IF			BMP_Err.top AND
			Level_masla_Norm.top AND
			T_masla_Norm.top AND
			Krans_ready_to_move.top AND
			Krans_Poloj.top AND
			Net_AO_KC_SHKS04M.top AND
			Avt_SHU_vkl.top AND
			Nalichie220_SHU_Ai.top AND
			BP_Norm.top AND
			Naprajenie_U_IM.top AND
			//NOTAnalogNS.top AND 
			Not_AS.top AND
			dP_kr1.top AND
			Auto_Rej.top AND
			Impuls_Gaz.top AND ((algmanager.mode=modegpa.MODE_PUSKAP_R) OR (algmanager.mode=modegpa.MODE_PUSKPP_R) OR 
								(algmanager.mode=modegpa.MODE_PUSKAP_Ch) OR (algmanager.mode=modegpa.MODE_PUSKPP_Ch) OR
								(algmanager.mode=modegpa.MODE_I) OR (algmanager.mode=modegpa.MODE_PUSKK)) THEN
								ppuThird:=TRUE; ELSE ppuThird:=FALSE;	END_IF//ППУ для третьего этапа пуска
			

	IF		(NOT (im.kran6.so OR im.kran6.sz OR
			im.kran4.so OR im.kran4.sz)) AND
			(Im.kran6.onStatus=statusDualInput.STATUS_ON) AND 
			(Im.kran4.onStatus=statusDualInput.STATUS_ON) AND 
			Net_AO_KC_SHKS04M.top AND (NOT remont ()) AND
			(Im.kran1.onStatus=statusDualInput.STATUS_On) AND
			(Im.kran2.onStatus=statusDualInput.STATUS_On) AND
			Impuls_Gaz.top AND ((algmanager.mode=modegpa.MODE_PUSKAP_R) OR (algmanager.mode=modegpa.MODE_PUSKPP_R) OR 
								(algmanager.mode=modegpa.MODE_PUSKAP_Ch) OR (algmanager.mode=modegpa.MODE_PUSKPP_Ch) OR
								(algmanager.mode=modegpa.MODE_I) OR (algmanager.mode=modegpa.MODE_PUSKK)) THEN
								ppuForth:=TRUE; ELSE ppuForth:=FALSE; END_IF	//ППУ для четвертого этапа пуска

METHOD PUBLIC Neisp_DI : BOOL
VAR_INPUT
END_VAR
Neisp_DI:= 
		((ystavki.dPmg_Rassogl.status = 1) OR
		im.NalichieBP1_NS.Q OR
		im.NalichieBP2_NS.Q OR
		im.NalichieBP3_NS.Q OR
		im.NalichieBP4_NS.Q OR
		im.NalichieBP5_NS.Q OR
		im.NalichieBP6_NS.Q OR
		im.NalichieBP7_BP8_NS.Q OR
		im.NalichieBP9_BP10_NS.Q OR
		im.Nalichie_CU_MV_NS.Q OR
		im.Nalichie220BEAO_NS.Q OR
		im.NalichiePer220naVhode_NS.Q OR
		im.NalichiePost220naVhode_NS.Q OR
		im.NalichieBP11_NS.Q OR
		im.NalichieBP12_NS.Q OR
		im.NET_U_PNS.Q OR
		im.NET_U_CMN.Q OR
		im.NET_U_NU1.Q OR
		im.NET_U_NU2.Q OR
 		im.kran1.sdvig OR
		im.kran2.sdvig OR
		im.kran3.sdvig OR
		im.kran3b.sdvig OR
		im.kran4.sdvig OR
		im.kran5.sdvig OR
		im.kran6.sdvig OR
		(im.LevelMaslaAkkum.status = 1) OR
		im.MainRegOff.Q OR
		im.AVR_Vozb_Malfanctional.Q OR
		im.AsynchronnyHod.Q);
END_METHOD

METHOD PUBLIC analogsNs : BOOL
VAR_INPUT
END_VAR
VAR
		
END_VAR
SUPER^();
analogsNs:=
	
		(ai.TStalisStatoraKanall.interval 											< statusAi.NORMAL) 	OR
		(ai.TStalisStatoraKanal2.interval 											< statusAi.NORMAL) 	OR
		(ai.TStalisStatoraKanal3.interval 											< statusAi.NORMAL) 	OR
		(ai.TMediStatoraKanall.interval 											< statusAi.NORMAL) 	OR
		(ai.TMediStatoraKanal2.interval 											< statusAi.NORMAL) 	OR
		(ai.TMediStatoraKanal3.interval 											< statusAi.NORMAL) 	OR
		(ai.TOpornogoPodshipnikaEDT_1.interval 										< statusAi.NORMAL) 	OR
		(ai.TOpornoYpornogoPodshipnikaEDT_2.interval 								< statusAi.NORMAL) 	OR
		(ai.TOpornoYpornogoPodshipnikaKolesaRedEDT_3.interval 						< statusAi.NORMAL) 	OR
		(ai.TOpornoYpornogoPodshipnikaKolesaRedHT_4.interval 						< statusAi.NORMAL) 	OR
		(ai.TOpornogoPodshipnikaShesterniReduktoraT_5.interval 						< statusAi.NORMAL) 	OR
		(ai.TOpornogoPodshipnikaReduktoraHT_6.interval 								< statusAi.NORMAL) 	OR
		(ai.TOpornoYpornogoPodshipnikaNagnetateljaT_7_1.interval 					< statusAi.NORMAL) 	OR
		(ai.TOpornoYpornogoPodshipnikaNagnetateljaT_7_2.interval 					< statusAi.NORMAL) 	OR
		(ai.TOpornoYpornogoPodshipnikaSvobodnogoKoncaNT_8_1.interval 				< statusAi.NORMAL) 	OR
		(ai.TOpornoYpornogoPodshipnikaSvobodnogoKoncaNT_8_2.interval 				< statusAi.NORMAL) 	OR
		(ai.TYpornogoPodshipnikaRavKolodokHT_9_1.interval 							< statusAi.NORMAL) 	OR
		(ai.TYpornogoPodshipnikaRavKolodokHT_9_2.interval 							< statusAi.NORMAL) 	OR
		(ai.TYpornogoPodshipnikaNerabKolodokHT_10_1.interval 						< statusAi.NORMAL) 	OR
		(ai.TYpornogoPodshipnikaNerabKolodokHT_10_2.interval 						< statusAi.NORMAL) 	OR
		(ai.THolodnogoVozduhaEDKanall.interval 										< statusAi.NORMAL) 	OR
		(ai.THolodnogoVozduhaEDKanal2.interval 										< statusAi.NORMAL) 	OR
		(ai.TGorjachegoVozduhaEDKanall.interval 									< statusAi.NORMAL) 	OR
		(ai.TGorjachegoVozduhaEDKanal2.interval 									< statusAi.NORMAL) 	OR
		(ai.TgazaNaVhodeH.interval 													< statusAi.NORMAL) 	OR
		(ai.TgazaNaVyhodeH.interval 												< statusAi.NORMAL) 	OR
		(ai.TMasladoAVOM.interval 													< statusAi.NORMAL) 	OR
		(ai.TMaslaPosleAVOM.interval 												< statusAi.NORMAL) 	OR
		(ai.TMaslaMB.interval 														< statusAi.NORMAL) 	OR
		(ai.TMaslaMB_TEN.interval 													< statusAi.NORMAL) 	OR
		(ai.DavlenijaMasloSmNizkoe.interval 										< statusAi.NORMAL) 	OR
		(ai.PerepadDavlenieNaMasloFiltre.interval 									< statusAi.NORMAL) 	OR
		(ai.DavlenijaMasloSmVysokoe.interval 										< statusAi.NORMAL) 	OR
		(ai.DavlenijaMaslaPosleGNS.interval 										< statusAi.NORMAL) 	OR
		(ai.DavlenijaMaslaPosleNU.interval 											< statusAi.NORMAL) 	OR
		(ai.PerepadDavlenieNaKonfuzore.interval 									< statusAi.NORMAL) 	OR
		(ai.OsSdvigNagnetatelja_Plus.interval 										< statusAi.NORMAL) 	OR
		(ai.OsSdvigNagnetatelja_Minus.interval 										< statusAi.NORMAL) 	OR
		(ai.PerepadDavlenieMasloGaz.interval 										< statusAi.NORMAL) 	OR
		(ai.DGazaNaVhodeNagnetatelja.interval 										< statusAi.NORMAL) 	OR
		(ai.DGazaNaVyhodeNagnetatelja.interval 										< statusAi.NORMAL) 	OR
		(ai.DavlenieImpulsGaz.interval 												< statusAi.NORMAL) 	OR
		(ai.YrovenMaslaMB.interval 													< statusAi.NORMAL) 	OR
		(ai.Kontrol_per220V.interval 												< statusAi.NORMAL) 	OR
		(ai.Kontrol_post220V.interval 												< statusAi.NORMAL) 	OR
		(ai.VibroSkorostOPED_T1.interval 											< statusAi.NORMAL) 	OR
		(ai.VibroSkorostOYPED_T2.interval 											< statusAi.NORMAL) 	OR
		(ai.VibroSkorostOYPKolesaED_T3.interval 									< statusAi.NORMAL) 	OR
		(ai.VibroSkorostOPKolesaRH_T4.interval 										< statusAi.NORMAL) 	OR
		(ai.VibroSkorostOPShesterniRED_T5.interval 									< statusAi.NORMAL) 	OR
		(ai.VibroSkorostOPShesterniReduktoraH_T6.interval 							< statusAi.NORMAL) 	OR
		(ai.TokStatora.interval 													< statusAi.NORMAL) ;
END_METHOD

METHOD PRIVATE AS_PS_Anologs : BOOL
VAR_INPUT
END_VAR

 AS_PS_Anologs:= 	(ai.TMediStatoraKanall.interval 								= statusAi.NORMAL) 	AND 
 				 	(ai.TMediStatoraKanal2.interval 								= statusAi.NORMAL) 	AND
				 	(ai.TMediStatoraKanal3.interval 								= statusAi.NORMAL) 	AND
				 	(ai.TStalisStatoraKanall.interval 								= statusAi.NORMAL) 	AND
				 	(ai.TStalisStatoraKanal2.interval 								= statusAi.NORMAL) 	AND
				 	(ai.TStalisStatoraKanal3.interval 								= statusAi.NORMAL) 	AND
				 	(ai.TGorjachegoVozduhaEDKanall.interval 						= statusAi.NORMAL) 	AND
				 	(ai.TGorjachegoVozduhaEDKanal2.interval 						= statusAi.NORMAL) 	AND
				 	(ai.THolodnogoVozduhaEDKanall.interval 							= statusAi.NORMAL) 	AND
				 	(ai.THolodnogoVozduhaEDKanal2.interval 							= statusAi.NORMAL) 	AND
				 	(ai.TOpornogoPodshipnikaEDT_1.interval 							= statusAi.NORMAL) 	AND
					(ai.TOpornoYpornogoPodshipnikaEDT_2.interval 					= statusAi.NORMAL) 	AND
					(ai.TOpornoYpornogoPodshipnikaKolesaRedEDT_3.interval 			= statusAi.NORMAL) 	AND
					(ai.TOpornoYpornogoPodshipnikaKolesaRedHT_4.interval 			= statusAi.NORMAL) 	AND
					(ai.TOpornogoPodshipnikaShesterniReduktoraT_5.interval 			= statusAi.NORMAL) 	AND
					(ai.TOpornogoPodshipnikaReduktoraHT_6.interval 					= statusAi.NORMAL) 	AND
					(ai.TOpornoYpornogoPodshipnikaNagnetateljaT_7_1.interval 		= statusAi.NORMAL) 	AND
					(ai.TOpornoYpornogoPodshipnikaNagnetateljaT_7_2.interval 		= statusAi.NORMAL) 	AND
					(ai.TOpornoYpornogoPodshipnikaSvobodnogoKoncaNT_8_1.interval 	= statusAi.NORMAL) 	AND
					(ai.TOpornoYpornogoPodshipnikaSvobodnogoKoncaNT_8_2.interval 	= statusAi.NORMAL) 	AND
					(ai.TYpornogoPodshipnikaRavKolodokHT_9_1.interval 				= statusAi.NORMAL) 	AND
					(ai.TYpornogoPodshipnikaRavKolodokHT_9_2.interval 				= statusAi.NORMAL) 	AND
					(ai.TYpornogoPodshipnikaNerabKolodokHT_10_1.interval 			= statusAi.NORMAL) 	AND
					(ai.TYpornogoPodshipnikaNerabKolodokHT_10_2.interval 			= statusAi.NORMAL) 	AND
					(ai.TgazaNaVhodeH.interval 										= statusAi.NORMAL) 	AND
					(ai.TgazaNaVyhodeH.interval 									= statusAi.NORMAL) 	AND
					(ai.TMasladoAVOM.interval 										= statusAi.NORMAL) 	AND
					(ai.TMaslaPosleAVOM.interval 									= statusAi.NORMAL) 	AND
					(ai.TMaslaMB.interval 											= statusAi.NORMAL) 	AND
					(ai.TMaslaMB_TEN.interval 										= statusAi.NORMAL) 	AND			
					(ai.VibroSkorostOPED_T1.interval 								= statusAi.NORMAL) 	AND
					(ai.VibroSkorostOYPED_T2.interval 								= statusAi.NORMAL) 	AND
					(ai.VibroSkorostOYPKolesaED_T3.interval 						= statusAi.NORMAL) 	AND
					(ai.VibroSkorostOPKolesaRH_T4.interval 							= statusAi.NORMAL) 	AND
					(ai.VibroSkorostOPShesterniRED_T5.interval 						= statusAi.NORMAL) 	AND
					(ai.VibroSkorostOPShesterniReduktoraH_T6.interval 				= statusAi.NORMAL) 	AND
					(ai.OsSdvigNagnetatelja_Plus.interval 							= statusAi.NORMAL) 	AND
					(ai.OsSdvigNagnetatelja_Minus.interval 							= statusAi.NORMAL);
END_METHOD

METHOD PRIVATE haveAlarms : BOOL
VAR_INPUT
	
END_VAR

haveAlarms:= (NOT (Im.AOKC_SHKC.Q)) AND (im.AOKC_SHKC_CK.status = 1);
END_METHOD

METHOD PUBLIC reset
VAR_INPUT
END_VAR
SUPER^.reset();
ppuFirst_for_Pusk_Ch:=FALSE;
ppuFirst_for_Pusk_R:=FALSE;
ppuFirst_for_V_Ch:=FALSE;
ppuFirst_for_V_R:=FALSE;
ppuFirst_for_Pms_dPmg:=FALSE;
ppuFirst_for_K:=FALSE;
ppuFirst_for_I:=FALSE;
ppuSecond_V_Pusk_Ch:=FALSE;
ppuSecond_V_Pusk_R:=FALSE;
ppuSecond_I:=FALSE;
ppuThird:=FALSE;
ppuForth:=FALSE;
statusSet.setBit(15,FALSE); //к пуску готов
statusSet.setBit(16, FALSE); //к проверкам готов
statusSet.setBit(17,FALSE); //ко 2-му этапу пуска готов
statusSet.setBit(18,FALSE); //ко 3-му этапу пуска готов
statusSet.setBit(19,FALSE); //к 4-му этапу пуска готов
statusSet.setBit(20,FALSE); //к 4-му этапу пуска готов
END_METHOD

METHOD PUBLIC writeImStatus
VAR_INPUT
END_VAR
SUPER^.writeImStatus();

statusSet.setBit(15,ppuFirst_for_Pusk_Ch); //к пуску частотному
statusSet.setBit(16,ppuFirst_for_Pusk_r); //к пуску реакторному
statusSet.setBit(17,(ppuFirst_for_V_Ch OR ppuFirst_for_V_r OR ppuFirst_for_Pms_dPmg OR ppuFirst_for_K OR ppuFirst_for_I)); //к проверкам готов
statusSet.setBit(18,(ppuSecond_V_Pusk_ch OR ppuSecond_V_Pusk_r OR ppuSecond_I)); //ко 2-му этапу пуска готов
statusSet.setBit(19,(ppuThird)); //к 3-му этапу пуска готов
statusSet.setBit(20,(ppuForth)); //к 4-му этапу пуска готов
END_METHOD

METHOD public CK_Di : BOOL
VAR_INPUT
END_VAR

 CK_Di:=	(im.PerepadDavlenieMasloGaz_CK.status = 1)	AND
 			(im.PerepadDavlenieKran1_CK.status = 1)		AND
			(im.LevelMaslaAkkum_CK.status = 1)			AND
			(im.LoadDriveisGranted_CK.status = 1)		AND
			(im.VozbutetelisReady_CK.status = 1)			AND
			(im.RegVozbOff_CK.status = 1)				AND
			(im.MainRegOff_CK.status = 1)				AND
			(im.AVR_Vozb_Malfanctional_CK.status = 1)		AND
			(im.OFFAvarSwitch_CK.status = 1)				AND
			(im.AsynchronnyHod_CK.status = 1)		AND
			(im.Avtomat_SHU_on_CK.status = 1)		AND
			(im.Avtomat_SHP_on_CK.status = 1)			AND
			(im.U_Sekcii_CK.status = 1)					AND
			(im.Reactorni_Pusk_CK.status = 1)				AND
			(im.Chastotniy_Pusk_CK.status = 1)			AND
			(im.Fail_Chastotniy_Pusk_CK.status = 1)		AND
			(im.Hand_Reg_rej_CK.status = 1)				AND
			(im.AOKC_SHKC_CK.status = 1)					AND
			(im.NO_fromSHU_CK.status = 1)					AND
			(im.AO_fromSHU_CK.status = 1)					AND
			(im.AO_PRU_CK.status = 1)						AND
			(im.NKU_1_On_CK.status = 1)					AND
			(im.NKU_2_On_CK.status = 1)					AND
			(im.MVvkl_NAlichie_CK.status = 1)				AND
			(im.MVvykl_NAlichie_CK.status = 1)			AND
			(im.MVControl_Work_NAlichie_CK.status = 1)		AND
			(im.PNS_vkl_NAlichie_CK.status = 1)			AND
			(im.NU1_vkl_NAlichie_CK.status = 1)			AND
			(im.NU2_vkl_NAlichie_CK.status = 1)			AND
			(im.AVOM1_vkl_NAlichie_CK.status = 1)			AND
			(im.AVOM2_vkl_NAlichie_CK.status = 1)			AND
			(im.AVOM3_vkl_NAlichie_CK.status = 1)			AND
			(im.AVOM4_vkl_NAlichie_CK.status = 1)			AND
			(im.TEN_MB_vkl_NAlichie_CK.status = 1)			AND
			(im.TEN_Kollectora_vkl_NAlichie_CK.status = 1)	AND
			(im.Kalorifer_AVOM_vkl_NAlichie_CK.status = 1)	AND
			(im.CMN_vkl_NAlichie_CK.status = 1) AND (im.kran1.onstatus<>statusDualInput.STATUS_ERROR)
			AND (im.kran2.onstatus<>statusDualInput.STATUS_ERROR) AND (im.kran3.onstatus<>statusDualInput.STATUS_ERROR)
			AND (im.kran3b.onstatus<>statusDualInput.STATUS_ERROR) AND (im.kran4.onstatus<>statusDualInput.STATUS_ERROR)
			AND (im.kran5.onstatus<>statusDualInput.STATUS_ERROR)	AND (im.kran6.onstatus<>statusDualInput.STATUS_ERROR);
END_METHOD

METHOD PUBLIC Remont : BOOL
VAR_INPUT
END_VAR
Remont := protections.p_TOpornogoPodshipnikaEDT_1.remont OR

	
		
		protections.p_TOpornoYpornogoPodshipnikaEDT_2.remont OR
		protections.p_TOpornoYpornogoPodshipnikaKolesaRedEDT_3.remont OR
		protections.p_TOpornoYpornogoPodshipnikaKolesaRedHT_4.remont OR
		protections.p_TOpornogoPodshipnikaShesterniReduktoraT_5.remont OR
		protections.p_TOpornogoPodshipnikaReduktoraHT_6.remont OR
		protections.p_TOpornoYpornogoPodshipnikaNagnetateljaT_7.remont OR
		protections.p_TOpornoYpornogoPodshipnikaSvobodnogoKoncaNT_8.remont OR
		protections.p_TYpornogoPodshipnikaRavKolodokHT_9.remont OR
		protections.p_TYpornogoPodshipnikaNerabKolodokHT_10.remont OR
		protections.p_TgazaNaVyhodeH.remont OR
		
	(*Давления*)
		
		protections.p_OsSdvigNagnetatelja_Plus.remont OR
		protections.p_OsSdvigNagnetatelja_Minus.remont OR
		protections.p_DGazaNaVhodeNagnetatelja_GPA_STOP.remont OR
		protections.p_DGazaNaVyhodeNagnetatelja_GPA_STOP.remont OR
		//protections.p_DGazaNaVhodeNagnetatelja.remont OR
		protections.p_DGazaNaVyhodeNagnetatelja.remont OR
		protections.p_PerepadDavlenieMasloGaz.remont OR
		protections.p_DavlenijaMasloSmNizkoe.remont OR
		protections.p_DavlenijaMasloSmVysokoe.remont OR
	
	(*Вибрация*)
		
		protections.p_VibroSkorostOPED_T1.remont OR
		protections.p_VibroSkorostOYPED_T2.remont OR
		protections.p_VibroSkorostOYPKolesaED_T3.remont OR
		protections.p_VibroSkorostOPKolesaRH_T4.remont OR
		protections.p_VibroSkorostOPShesterniRED_T5.remont OR
		protections.p_VibroSkorostOPShesterniReduktoraH_T6.remont OR
	(*Дискретные сигналы *)
		
		protections.p_PerepadDavlenieMasloGaz_Less100.remont OR
		protections.p_RegVozbOff.remont OR
		protections.p_Fail_Chastotniy_Pusk.remont OR
		protections.p_OFFAvarSwitch.remont OR
		protections.p_AOKC_SHKC.remont OR
		protections.p_AO_PRU.remont OR
		protections.p_AO_fromSHU.remont OR	
					
(*Защиты по ИМ *)																							
		protections.p_mvOff.remont OR
		protections.p_kran1.remont OR
		protections.p_kran2.remont;
END_METHOD

END_FUNCTION_BLOCK

// K1/std12k5/Pusk/puskFirst_faza1
	{attribute 'symbol' := 'none'}
FUNCTION_BLOCK puskFirst_faza1 EXTENDS StepBySteapAlgoritm
VAR_INPUT
	
END_VAR
VAR_OUTPUT
END_VAR
VAR
	{attribute 'symbol' := 'read'}
	timer240:		ph_Timer (table:=ADR(phasesTable)):=		(phaseNumber:=0, delay:=T#240S);
	pnsOn:			ph_Switch (table:=ADR(phasesTable)):=		(phaseNumber:=1, Im:=Im.pns, act:=DualStateImAction.on);
	psmMore50:		CustomPhase (table:=ADR(phasesTable)):=		(phaseNumber:=2);
	psmMore300:		CustomPhase (table:=ADR(phasesTable)):=		(phaseNumber:=3);
	Protection_Pms: CustomPhase (table:=ADR(phasesTable)):=		(phaseNumber:=4);
	Error_Alg:		CustomPhase (table:=ADR(phasesTable)):=		(phaseNumber:=5);
END_VAR

SUPER^();
IF 	NOT Protection_Pms.top THEN
	timer240.run (); //запускаем таймер включаем ПНС
END_IF;
IF NOT pnsON.start THEN
	pnsOn.run();
END_IF
///////////////////////////////////////////////////////
IF 	pnsOn.top THEN //ПНС включен и таймер не истек
	psmMore50.run(); //запускаем проверку условия Pмс >50 
	psmMore300.run(); //запускаем проверку условия Pмс >300 
END_IF
///////////////////////////////////////////////////////
IF	psmMore50.start AND (NOT psmMore50.top) THEN
	IF 	ai.DavlenijaMasloSmNizkoe.interval>=statusAi.NORMAL AND ai.DavlenijaMasloSmNizkoe.value > 50  THEN
	  	psmMore50.top:=TRUE;
	END_IF
END_IF
///////////////////////////////////////////////////////
IF  psmMore300.start AND (NOT psmMore300.top) THEN
	IF 	ai.DavlenijaMasloSmVysokoe.interval>=statusAi.NORMAL AND ai.DavlenijaMasloSmVysokoe.value > 300  THEN
	  	psmMore300.top:=TRUE;
	END_IF	
END_IF
///////////////////////////////////////////////////////
IF	psmMore50.top AND psmMore300.top THEN
	Protection_Pms.run ();
END_IF
///////////////////////////////////////////////////////
IF	Protection_Pms.start AND (NOT Protection_Pms.top) THEN //защита по давлению масла смазки включить
	protections.p_DavlenijaMasloSmNizkoe.run();
	protections.p_DavlenijaMasloSmVysokoe.run ();
	Protection_Pms.top := TRUE;
END_IF
///////////////////////////////////////////////////////
IF	timer240.top THEN //Ошибка завершения алгоритма по таймеру
	Error_Alg.ERROR := TRUE;
ELSE
	Error_Alg.ERROR := FALSE;	
END_IF
///////////////////////////////////////////////////////
IF	Protection_Pms.top THEN
	timer240.reset();
	end ();
END_IF
///////////////////////////////////////////////////////

METHOD PUBLIC reset
VAR_INPUT
END_VAR
SUPER^.reset();
statusSet.setBit(15,0);
END_METHOD

METHOD PUBLIC run
VAR_INPUT
END_VAR
SUPER^.run();
statusSet.setBit(15,1);
END_METHOD

END_FUNCTION_BLOCK

// K2/std12k5/Pusk/puskFirst_faza1
	{attribute 'symbol' := 'none'}
FUNCTION_BLOCK puskFirst_faza1 EXTENDS StepBySteapAlgoritm
VAR_INPUT
	
END_VAR
VAR_OUTPUT
END_VAR
VAR
	{attribute 'symbol' := 'read'}
	timer240:		ph_Timer (table:=ADR(phasesTable)):=		(phaseNumber:=0, delay:=T#240S);
	pnsOn:			ph_Switch (table:=ADR(phasesTable)):=		(phaseNumber:=1, Im:=Im.pns, act:=DualStateImAction.on);
	psmMore50:		CustomPhase (table:=ADR(phasesTable)):=		(phaseNumber:=2);
	psmMore300:		CustomPhase (table:=ADR(phasesTable)):=		(phaseNumber:=3);
	Protection_Pms: CustomPhase (table:=ADR(phasesTable)):=		(phaseNumber:=4);
	Error_Alg:		CustomPhase (table:=ADR(phasesTable)):=		(phaseNumber:=5);
END_VAR

SUPER^();
IF 	NOT Protection_Pms.top THEN
	timer240.run (); //запускаем таймер включаем ПНС
END_IF;
IF NOT pnsON.start THEN
	pnsOn.run();
END_IF
///////////////////////////////////////////////////////
IF 	pnsOn.top THEN //ПНС включен и таймер не истек
	psmMore50.run(); //запускаем проверку условия Pмс >50 
	psmMore300.run(); //запускаем проверку условия Pмс >300 
END_IF
///////////////////////////////////////////////////////
IF	psmMore50.start AND (NOT psmMore50.top) THEN
	IF 	ai.DavlenijaMasloSmNizkoe.interval>=statusAi.NORMAL AND ai.DavlenijaMasloSmNizkoe.value > 50  THEN
	  	psmMore50.top:=TRUE;
	END_IF
END_IF
///////////////////////////////////////////////////////
IF  psmMore300.start AND (NOT psmMore300.top) THEN
	IF 	ai.DavlenijaMasloSmVysokoe.interval>=statusAi.NORMAL AND ai.DavlenijaMasloSmVysokoe.value > 300  THEN
	  	psmMore300.top:=TRUE;
	END_IF	
END_IF
///////////////////////////////////////////////////////
IF	psmMore50.top AND psmMore300.top THEN
	Protection_Pms.run ();
END_IF
///////////////////////////////////////////////////////
IF	Protection_Pms.start AND (NOT Protection_Pms.top) THEN //защита по давлению масла смазки включить
	protections.p_DavlenijaMasloSmNizkoe.run();
	protections.p_DavlenijaMasloSmVysokoe.run ();
	Protection_Pms.top := TRUE;
END_IF
///////////////////////////////////////////////////////
IF	timer240.top THEN //Ошибка завершения алгоритма по таймеру
	Error_Alg.ERROR := TRUE;
ELSE
	Error_Alg.ERROR := FALSE;	
END_IF
///////////////////////////////////////////////////////
IF	Protection_Pms.top THEN
	timer240.reset();
	end ();
END_IF
///////////////////////////////////////////////////////

METHOD PUBLIC reset
VAR_INPUT
END_VAR
SUPER^.reset();
statusSet.setBit(15,0);
END_METHOD

METHOD PUBLIC run
VAR_INPUT
END_VAR
SUPER^.run();
statusSet.setBit(15,1);
END_METHOD

END_FUNCTION_BLOCK

// K1/std12k5/Pusk/puskFirst_faza2
	{attribute 'symbol' := 'none'}
FUNCTION_BLOCK puskFirst_faza2 EXTENDS StepBySteapAlgoritm
VAR_INPUT
	
END_VAR
VAR_OUTPUT
END_VAR
VAR
	{attribute 'symbol' := 'read'}
	timer240:		ph_Timer 	(table:=ADR(phasesTable)):=		(phaseNumber:=0, delay:=T#240S);
	nuOn:			CustomPhase (table:=ADR(phasesTable)):=		(phaseNumber:=1);
	dPmg_more100:	CustomPhase (table:=ADR(phasesTable)):=		(phaseNumber:=2);
	Error_Alg:		CustomPhase (table:=ADR(phasesTable)):=		(phaseNumber:=3);
	Auto_NU1:		CustomPhase (table:=ADR(phasesTable)):=		(phaseNumber:=4);
END_VAR

SUPER^();
IF 	NOT dPmg_more100.top THEN
	timer240.run (); //запускаем таймер включаем ПНС
END_IF
IF	NOT nuon.start THEN
	nuOn.run();
END_IF
///////////////////////////////////////////////////////
IF 	nuOn.start AND NOT nuOn.top THEN //НУ включен
	CASE 	im.nu.mainNasos.Value OF
	0:		im.nu.nu1.on ();
	1:		im.nu.nu2.on ();
	END_CASE
END_IF
///////////////////////////////////////////////////////
IF	((im.nu.nu1.onStatus = statusDualInput.status_on) OR (im.nu.nu2.onStatus = statusDualInput.status_on)) AND  nuOn.start THEN
	dPmg_more100.run(); //запускаем проверку условия dPmg_more100
	nuOn.top:=TRUE;
END_IF
///////////////////////////////////////////////////////
IF	dPmg_more100.start AND (NOT dPmg_more100.top) THEN
	IF 	(NOT im.PerepadDavlenieMasloGaz_Less100.Q) AND (im.PerepadDavlenieMasloGaz_CK.status = 1) AND 
		(ai.PerepadDavlenieMasloGaz.interval	>=	statusAi.NORMAL) AND (ai.PerepadDavlenieMasloGaz.value > 150) THEN
	  	dPmg_more100.top:=TRUE;
	END_IF
END_IF
///////////////////////////////////////////////////////
IF	timer240.top THEN //Ошибка завершения алгоритма по таймеру
	Error_Alg.ERROR := TRUE;
ELSE
	Error_Alg.ERROR := FALSE;	
END_IF
///////////////////////////////////////////////////////
IF	dPmg_more100.top AND nuOn.top THEN
	Auto_NU1.top:=TRUE;
	protections.p_PerepadDavlenieMasloGaz.run();
	protections.p_PerepadDavlenieMasloGaz_Less100.run ();
	protections.p_DGazaNaVhodeNagnetatelja_GPA_STOP.reset ();
	protections.p_DGazaNaVyhodeNagnetatelja_GPA_STOP.reset ();
	algoritms.autoNu_1.CanRun:=TRUE;
	algoritms.autoNu_1.run ();
	timer240.reset();
	end();
END_IF

END_FUNCTION_BLOCK

// K2/std12k5/Pusk/puskFirst_faza2
	{attribute 'symbol' := 'none'}
FUNCTION_BLOCK puskFirst_faza2 EXTENDS StepBySteapAlgoritm
VAR_INPUT
	
END_VAR
VAR_OUTPUT
END_VAR
VAR
	{attribute 'symbol' := 'read'}
	timer240:		ph_Timer 	(table:=ADR(phasesTable)):=		(phaseNumber:=0, delay:=T#240S);
	nuOn:			CustomPhase (table:=ADR(phasesTable)):=		(phaseNumber:=1);
	dPmg_more100:	CustomPhase (table:=ADR(phasesTable)):=		(phaseNumber:=2);
	Error_Alg:		CustomPhase (table:=ADR(phasesTable)):=		(phaseNumber:=3);
	Auto_NU1:		CustomPhase (table:=ADR(phasesTable)):=		(phaseNumber:=4);
END_VAR

SUPER^();
IF 	NOT dPmg_more100.top THEN
	timer240.run (); //запускаем таймер включаем ПНС
END_IF;
IF	NOT nuon.start THEN
	nuOn.run();
END_IF
///////////////////////////////////////////////////////
IF 	nuOn.start AND NOT nuOn.top THEN //НУ включен
	CASE 	im.nu.mainNasos.Value OF
	0:		im.nu.nu1.on ();
	1:		im.nu.nu2.on ();
	END_CASE
END_IF
///////////////////////////////////////////////////////
IF	((im.nu.nu1.onStatus = statusDualInput.status_on) OR (im.nu.nu2.onStatus = statusDualInput.status_on)) AND  nuOn.start THEN
	dPmg_more100.run(); //запускаем проверку условия dPmg_more100
	nuOn.top:=TRUE;
END_IF
///////////////////////////////////////////////////////
IF	dPmg_more100.start AND (NOT dPmg_more100.top) THEN
	IF 	(NOT im.PerepadDavlenieMasloGaz_Less100.Q) AND (im.PerepadDavlenieMasloGaz_CK.status = 1) AND 
		(ai.PerepadDavlenieMasloGaz.interval	>=	statusAi.NORMAL) AND (ai.PerepadDavlenieMasloGaz.value > 150) THEN
	  	dPmg_more100.top:=TRUE;
	END_IF
END_IF
///////////////////////////////////////////////////////
IF	timer240.top THEN //Ошибка завершения алгоритма по таймеру
	Error_Alg.ERROR := TRUE;
ELSE
	Error_Alg.ERROR := FALSE;	
END_IF
///////////////////////////////////////////////////////
IF	dPmg_more100.top AND nuOn.top THEN
	Auto_NU1.top:=TRUE;
	protections.p_PerepadDavlenieMasloGaz.run();
	protections.p_PerepadDavlenieMasloGaz_Less100.run ();
	protections.p_DGazaNaVhodeNagnetatelja_GPA_STOP.reset ();
	protections.p_DGazaNaVyhodeNagnetatelja_GPA_STOP.reset ();
	algoritms.autoNu_1.CanRun:=TRUE;
	algoritms.autoNu_1.run ();
	timer240.reset();
	end();
END_IF

END_FUNCTION_BLOCK

// K1/std12k5/Pusk/puskSecond_faza_Reactor
{attribute 'symbol' := 'none'}
FUNCTION_BLOCK puskSecond_faza_Reactor EXTENDS StepBySteapAlgoritm
VAR_INPUT
	autoAVOM_canrun_flag:BOOL;
END_VAR
VAR_OUTPUT
	
END_VAR
VAR
	{attribute 'symbol' := 'read'}
	timer25:			ph_Timer (table:=ADR(phasesTable)):=		(phaseNumber:=0, delay:=T#25S);
	{attribute 'symbol' := 'read'}
	timer3:				ph_Timer (table:=ADR(phasesTable)):=		(phaseNumber:=1, delay:=T#3S);
	mvOn:				ph_Switch (table:=ADR(phasesTable)):=		(phaseNumber:=2, Im:=Im.mv, act:=DualStateImAction.on);
	pGNSmore04:			CustomPhase (table:=ADR(phasesTable)):=		(phaseNumber:=3);
	gotov_K_zagruzke: 	ph_SingleSignal (table:=ADR(phasesTable)):=	(phaseNumber:=4, im:=im.LoadDriveisGranted, expectedValue:=TRUE);
	
	dPmg_Top:			CustomPhase (table:=ADR(phasesTable)):=		(phaseNumber:=6);
	
	Mv_Error:			CustomPhase (table:=ADR(phasesTable)):=		(phaseNumber:=8);
	AutoPNS_start:		CustomPhase (table:=ADR(phasesTable)):=		(phaseNumber:=9);
END_VAR

SUPER^();
IF 	NOT mvOn.top THEN
	timer25.run (); //запускаем таймер 25 сек
END_IF
IF	NOT mvOn.top THEN
	timer3.run (); //запускаем таймер 3 сек
END_IF
IF	NOT mvOn.start THEN
	mvOn.run();
END_IF
///////////////////////////////////////////////////////
IF 	mvOn.top  THEN 
	IF	NOT pGNSmore04.start AND ((algManager.mode = modegpa.MODE_PUSKAP_R) OR (algManager.mode = modegpa.MODE_PUSKPP_R)) THEN //проверяем условие по давление за ГНС > 400 кПа
		pGNSmore04.run(); 
	END_IF
	IF	NOT autoAVOM_canrun_flag THEN
		algoritms.S_AutoAVOM.CanRun:=TRUE;
		autoAVOM_canrun_flag:=TRUE;
	END_IF
	timer3.reset ();
	timer25.reset ();
	Mv_Error.error := FALSE;
	gotov_K_zagruzke.run();
	IF	(NOT dPmg_Top.start) AND ((algManager.mode = modegpa.MODE_PUSKAP_R) OR (algManager.mode = modegpa.MODE_PUSKPP_R)) THEN
		dPmg_Top.run ();
	END_IF
	protections.p_mvOff.run (); //включаем защиты по МВ и возбудителю
	protections.p_OFFAvarSwitch.run();
	protections.p_RegVozbOff.run();
ELSIF	NOT mvOn.top AND timer3.top THEN
		Mv_Error.error := TRUE;
END_IF

///////////////////////////////////////////////////////
IF	dPmg_Top.start AND (NOT dPmg_Top.top) THEN
	IF	(NOT im.PerepadDavlenieMasloGaz_Less100.Q) AND (im.PerepadDavlenieMasloGaz_CK.status = 1) AND (ai.PerepadDavlenieMasloGaz.value > 150)	THEN //по аналогу проверяем только значение, т.к. при пуске может уйти в зашкал
		dPmg_Top.top:=TRUE;
		protections.p_PerepadDavlenieMasloGaz.run();
		protections.p_PerepadDavlenieMasloGaz_Less100.run ();
		protections.p_DGazaNaVhodeNagnetatelja_GPA_STOP.reset ();
		protections.p_DGazaNaVyhodeNagnetatelja_GPA_STOP.reset ();
		algoritms.autoNu_2.CanRun:=TRUE;
		algoritms.autoNu_2.run ();
	END_IF
END_IF
///////////////////////////////////////////////////////
IF	pGNSmore04.start AND (NOT pGNSmore04.top) THEN //Давление после ГНС больше 400 кПА
	IF 	(ai.DavlenijaMaslaPosleGNS.interval	>=statusAi.NORMAL) AND (ai.DavlenijaMaslaPosleGNS.value	 > 400) THEN
	  	pGNSmore04.top:=TRUE; 
	END_IF
END_IF
///////////////////////////////////////////////////////
IF	((pGNSmore04.top AND gotov_K_zagruzke.top AND dPmg_Top.top AND ((algManager.mode = modegpa.MODE_PUSKAP_R) OR (algManager.mode = modegpa.MODE_PUSKPP_R))) OR 
	(gotov_K_zagruzke.top AND ((algManager.mode = modegpa.MODE_PUSKV_R) OR (algManager.mode = modegpa.MODE_I)))) AND NOT AutoPNS_start.top  THEN 
	algoritms.AutoPNS_Start.CanRun :=TRUE;
	algoritms.AutoPNS_Start.run();
	AutoPNS_start.top:=TRUE;
	end();
END_IF
IF	timer25.top AND Mv_Error.error THEN
	algoritms.ao.CanRun:=TRUE;
	algoritms.ao.run ();
	
END_IF

METHOD PUBLIC reset
VAR_INPUT
END_VAR
SUPER^.reset();
statusSet.setBit(15,0);
END_METHOD

METHOD PUBLIC run
VAR_INPUT
END_VAR
SUPER^.run();
statusSet.setBit(15,1);
END_METHOD

END_FUNCTION_BLOCK

// K2/std12k5/Pusk/puskSecond_faza_Reactor
{attribute 'symbol' := 'none'}
FUNCTION_BLOCK puskSecond_faza_Reactor EXTENDS StepBySteapAlgoritm
VAR_INPUT
	autoAVOM_canrun_flag:BOOL;
END_VAR
VAR_OUTPUT
	
END_VAR
VAR
	{attribute 'symbol' := 'read'}
	timer25:			ph_Timer (table:=ADR(phasesTable)):=		(phaseNumber:=0, delay:=T#25S);
	{attribute 'symbol' := 'read'}
	timer3:				ph_Timer (table:=ADR(phasesTable)):=		(phaseNumber:=1, delay:=T#3S);
	mvOn:				ph_Switch (table:=ADR(phasesTable)):=		(phaseNumber:=2, Im:=Im.mv, act:=DualStateImAction.on);
	pGNSmore04:			CustomPhase (table:=ADR(phasesTable)):=		(phaseNumber:=3);
	gotov_K_zagruzke: 	ph_SingleSignal (table:=ADR(phasesTable)):=	(phaseNumber:=4, im:=im.LoadDriveisGranted, expectedValue:=TRUE);
	
	dPmg_Top:			CustomPhase (table:=ADR(phasesTable)):=		(phaseNumber:=6);
	
	Mv_Error:			CustomPhase (table:=ADR(phasesTable)):=		(phaseNumber:=8);
	AutoPNS_start:		CustomPhase (table:=ADR(phasesTable)):=		(phaseNumber:=9);
END_VAR

SUPER^();
IF 	NOT mvOn.top THEN
	timer25.run (); //запускаем таймер 25 сек
END_IF
IF	NOT mvOn.top THEN
	timer3.run (); //запускаем таймер 3 сек
END_IF
IF	NOT mvOn.start THEN
	mvOn.run();
END_IF
///////////////////////////////////////////////////////
IF 	mvOn.top  THEN 
	IF	NOT pGNSmore04.start AND ((algManager.mode = modegpa.MODE_PUSKAP_R) OR (algManager.mode = modegpa.MODE_PUSKPP_R)) THEN //проверяем условие по давление за ГНС > 400 кПа
		pGNSmore04.run(); 
	END_IF
	IF	NOT autoAVOM_canrun_flag THEN
		algoritms.S_AutoAVOM.CanRun:=TRUE;
		autoAVOM_canrun_flag:=TRUE;
	END_IF
	timer3.reset ();
	timer25.reset ();
	Mv_Error.error := FALSE;
	gotov_K_zagruzke.run();
	IF	(NOT dPmg_Top.start) AND ((algManager.mode = modegpa.MODE_PUSKAP_R) OR (algManager.mode = modegpa.MODE_PUSKPP_R)) THEN
		dPmg_Top.run ();
	END_IF
	protections.p_mvOff.run (); //включаем защиты по МВ и возбудителю
	protections.p_OFFAvarSwitch.run();
	protections.p_RegVozbOff.run();
ELSIF	NOT mvOn.top AND timer3.top THEN
		Mv_Error.error := TRUE;
END_IF

///////////////////////////////////////////////////////
IF	dPmg_Top.start AND (NOT dPmg_Top.top) THEN
	IF	(NOT im.PerepadDavlenieMasloGaz_Less100.Q) AND (im.PerepadDavlenieMasloGaz_CK.status = 1)AND (ai.PerepadDavlenieMasloGaz.value > 150)	THEN //по аналогу проверяем только значение, т.к. при пуске может уйти в зашкал
		dPmg_Top.top:=TRUE;
		protections.p_PerepadDavlenieMasloGaz.run();
		protections.p_PerepadDavlenieMasloGaz_Less100.run ();
		protections.p_DGazaNaVhodeNagnetatelja_GPA_STOP.reset ();
		protections.p_DGazaNaVyhodeNagnetatelja_GPA_STOP.reset ();
		algoritms.autoNu_2.CanRun:=TRUE;
		algoritms.autoNu_2.run ();
	END_IF
END_IF
///////////////////////////////////////////////////////
IF	pGNSmore04.start AND (NOT pGNSmore04.top) THEN //Давление после ГНС больше 400 кПА
	IF 	(ai.DavlenijaMaslaPosleGNS.interval	>=statusAi.NORMAL) AND (ai.DavlenijaMaslaPosleGNS.value	 > 400) THEN
	  	pGNSmore04.top:=TRUE; 
	END_IF
END_IF
///////////////////////////////////////////////////////
IF	((pGNSmore04.top AND gotov_K_zagruzke.top AND dPmg_Top.top AND ((algManager.mode = modegpa.MODE_PUSKAP_R) OR (algManager.mode = modegpa.MODE_PUSKPP_R))) OR 
	(gotov_K_zagruzke.top AND ((algManager.mode = modegpa.MODE_PUSKV_R) OR (algManager.mode = modegpa.MODE_I)))) AND NOT AutoPNS_start.top  THEN 
	algoritms.AutoPNS_Start.CanRun :=TRUE;
	algoritms.AutoPNS_Start.run();
	AutoPNS_start.top:=TRUE;
	end();
END_IF
IF	timer25.top AND Mv_Error.error THEN
	algoritms.ao.CanRun:=TRUE;
	algoritms.ao.run ();
	
END_IF

METHOD PUBLIC reset
VAR_INPUT
END_VAR
SUPER^.reset();
statusSet.setBit(15,0);
END_METHOD

METHOD PUBLIC run
VAR_INPUT
END_VAR
SUPER^.run();
statusSet.setBit(15,1);
END_METHOD

END_FUNCTION_BLOCK

// K1/std12k5/Pusk/puskThird_faza
	{attribute 'symbol' := 'none'}
FUNCTION_BLOCK puskThird_faza EXTENDS StepBySteapAlgoritm
VAR_INPUT
	Smazka_1_2:BOOL;
END_VAR
VAR_OUTPUT
	
END_VAR
VAR
	{attribute 'symbol' := 'read'}
	timer480:		ph_Timer (table:=ADR(phasesTable)):=		(phaseNumber:=0, delay:=T#480S);
	kran4Open:		CustomPhase (table:=ADR(phasesTable)):=		(phaseNumber:=1);
	{attribute 'symbol' := 'read'}
	waitAfterKran4:	ph_Timer (table:=ADR(phasesTable)):=		(phaseNumber:=2, delay:=T#10S);
	kran5Close:		ph_Kran (table:=ADR(phasesTable)):=			(phaseNumber:=3, Im:=Im.kran5, act:=DualStateImAction.off);	
	kran3bOpen:		CustomPhase (table:=ADR(phasesTable)):=		(phaseNumber:=4);
	dP_kr1less100: 	ph_SingleSignal (table:=ADR(phasesTable)):=	(phaseNumber:=5, im:=Im.PerepadDavlenieKran1_Less100, expectedValue:=TRUE);
	Pvh_vyhMore5:	CustomPhase (table:=ADR(phasesTable)):=		(phaseNumber:=6);
	kran1Open:		ph_Kran (table:=ADR(phasesTable)):=			(phaseNumber:=7, Im:=Im.kran1, act:=DualStateImAction.on);	
	kran2Open:		ph_Kran (table:=ADR(phasesTable)):=			(phaseNumber:=8, Im:=Im.kran2, act:=DualStateImAction.on);
	kran3Open:		ph_Kran (table:=ADR(phasesTable)):=			(phaseNumber:=9, Im:=Im.kran3, act:=DualStateImAction.on);
	kran3bClose:	ph_Kran (table:=ADR(phasesTable)):=			(phaseNumber:=10, Im:=Im.kran3b, act:=DualStateImAction.off);
	Err_ALG:		CustomPhase (table:=ADR(phasesTable)):=		(phaseNumber:=11);
END_VAR

SUPER^();
IF	NOT (kran3bClose.top) THEN
	timer480.run (); //запускаем таймер 480 секунд
END_IF;
////////////////////***Открываем кран 4****//////////////////////////
IF	NOT kran1Open.top AND im.kran4._cmdreset.IN = FALSE  THEN
	
	im.Kr_4_Open_From_Alg.on();
	kran4Open.run();
END_IF;
IF	kran4Open.start AND NOT kran4Open.top THEN
	IF	im.kran4.onStatus = statusDualInput.STATUS_ON THEN
		kran4Open.top:=TRUE;
	END_IF
END_IF
///////////////////////////////////////////////////
IF 	kran4Open.top THEN //продувка 10 секунд
	waitAfterKran4.run();
END_IF
///////////////////////////////////////////////////
IF	waitAfterKran4.top THEN
	kran5Close.run(); //закрываем кран 5
END_IF
///////////////////////////////////////////////////
IF	kran5Close.top THEN//Если кран 5 зарыт, то
	kran3bOpen.run ();//Проверяем открытие крана  3б
	dP_kr1less100.run (); //и перепад на кране 1
	Pvh_vyhMore5.run();
END_IF
///////////////////////////////////////////////////
IF	Pvh_vyhMore5.start AND NOT Pvh_vyhMore5.top THEN //Давление газа на входе/выходе нагнетателя > 4 МПа
	IF	(ai.DGazaNaVhodeNagnetatelja.interval >=statusAi.NORMAL) AND (ai.DGazaNaVhodeNagnetatelja.value	 >= 4) AND 
		(ai.DGazaNaVyhodeNagnetatelja.interval >=statusAi.NORMAL) AND (ai.DGazaNaVyhodeNagnetatelja.value	 >= 4) THEN
		Pvh_vyhMore5.top := TRUE;
		//protections.p_DGazaNaVhodeNagnetatelja.run ();
		protections.p_DGazaNaVyhodeNagnetatelja.run ();
	END_IF;
END_IF
///////////////////////////////////////////////////
IF	kran3bOpen.start AND NOT kran3bOpen.top THEN//Проверяем, что открыт крана  3б
	IF	im.kran3b.onStatus=statusDualInput.STATUS_ON THEN
		kran3bOpen.top :=TRUE;	
	END_IF
END_IF
///////////////////////////////////////////////////
IF	kran3bOpen.top AND	kran5Close.top AND dP_kr1less100.top AND Pvh_vyhMore5.top THEN
	kran1Open.run ();  //кран 1 и 2 открываем
	kran2Open.run (); 
	kran3Open.run ();
	Smazka_1_2:=TRUE;
END_IF
IF	kran1Open.top THEN
	im.Kr_4_Open_From_Alg.off();
	ystavki.Block_kr4_alg.setValue (0);
END_IF
///////////////////////////////////////////////////
IF	kran1Open.top AND kran2Open.top AND kran3Open.top THEN //закрываем кран 3бис
	kran3bClose.run (); 
END_IF
///////////////////////////////////////////////////
IF 	kran3bClose.top THEN
	Err_ALG.error :=FALSE;
	timer480.reset ();
	end ();
ELSIF	(NOT (kran3bClose.top)) AND timer480.top THEN
		Err_ALG.error :=TRUE;
END_IF

METHOD PUBLIC reset
VAR_INPUT
END_VAR
SUPER^.reset();
im.Kr_4_Open_From_Alg.off();

statusSet.setBit(15,0);
END_METHOD

METHOD PUBLIC run
VAR_INPUT
END_VAR
SUPER^.run();
statusSet.setBit(15,1);
ystavki.Block_kr4_alg.setValue (1);
END_METHOD

END_FUNCTION_BLOCK

// K2/std12k5/Pusk/puskThird_faza
	{attribute 'symbol' := 'none'}
FUNCTION_BLOCK puskThird_faza EXTENDS StepBySteapAlgoritm
VAR_INPUT
	Smazka_1_2:BOOL;
END_VAR
VAR_OUTPUT
	
END_VAR
VAR
	{attribute 'symbol' := 'read'}
	timer480:		ph_Timer (table:=ADR(phasesTable)):=		(phaseNumber:=0, delay:=T#480S);
	kran4Open:		CustomPhase (table:=ADR(phasesTable)):=		(phaseNumber:=1);
	{attribute 'symbol' := 'read'}
	waitAfterKran4:	ph_Timer (table:=ADR(phasesTable)):=		(phaseNumber:=2, delay:=T#10S);
	kran5Close:		ph_Kran (table:=ADR(phasesTable)):=			(phaseNumber:=3, Im:=Im.kran5, act:=DualStateImAction.off);	
	kran3bOpen:		CustomPhase (table:=ADR(phasesTable)):=		(phaseNumber:=4);
	dP_kr1less100: 	ph_SingleSignal (table:=ADR(phasesTable)):=	(phaseNumber:=5, im:=Im.PerepadDavlenieKran1_Less100, expectedValue:=TRUE);
	Pvh_vyhMore5:	CustomPhase (table:=ADR(phasesTable)):=		(phaseNumber:=6);
	kran1Open:		ph_Kran (table:=ADR(phasesTable)):=			(phaseNumber:=7, Im:=Im.kran1, act:=DualStateImAction.on);	
	kran2Open:		ph_Kran (table:=ADR(phasesTable)):=			(phaseNumber:=8, Im:=Im.kran2, act:=DualStateImAction.on);
	kran3Open:		ph_Kran (table:=ADR(phasesTable)):=			(phaseNumber:=9, Im:=Im.kran3, act:=DualStateImAction.on);
	kran3bClose:	ph_Kran (table:=ADR(phasesTable)):=			(phaseNumber:=10, Im:=Im.kran3b, act:=DualStateImAction.off);
	Err_ALG:		CustomPhase (table:=ADR(phasesTable)):=		(phaseNumber:=11);
END_VAR

SUPER^();
IF	NOT (kran3bClose.top) THEN
	timer480.run (); //запускаем таймер 480 секунд
END_IF;
////////////////////***Открываем кран 4****//////////////////////////
IF	NOT kran1Open.top AND im.kran4._cmdreset.IN = FALSE  THEN

	im.Kr_4_Open_From_Alg.on();
	kran4Open.run();
END_IF;
IF	kran4Open.start AND NOT kran4Open.top THEN
	IF	im.kran4.onStatus = statusDualInput.STATUS_ON THEN
		kran4Open.top:=TRUE;
	END_IF
END_IF
///////////////////////////////////////////////////
IF 	kran4Open.top THEN //продувка 10 секунд
	waitAfterKran4.run();
END_IF
///////////////////////////////////////////////////
IF	waitAfterKran4.top THEN
	kran5Close.run(); //закрываем кран 5
END_IF
///////////////////////////////////////////////////
IF	kran5Close.top THEN//Если кран 5 зарыт, то
	kran3bOpen.run ();//Проверяем открытие крана  3б
	dP_kr1less100.run (); //и перепад на кране 1
	Pvh_vyhMore5.run();
END_IF
///////////////////////////////////////////////////
IF	Pvh_vyhMore5.start AND NOT Pvh_vyhMore5.top THEN //Давление газа на входе/выходе нагнетателя > 4 МПа
	IF	(ai.DGazaNaVhodeNagnetatelja.interval >=statusAi.NORMAL) AND (ai.DGazaNaVhodeNagnetatelja.value	 >= 4) AND 
		(ai.DGazaNaVyhodeNagnetatelja.interval >=statusAi.NORMAL) AND (ai.DGazaNaVyhodeNagnetatelja.value	 >= 4) THEN
		Pvh_vyhMore5.top := TRUE;
		//protections.p_DGazaNaVhodeNagnetatelja.run ();
		protections.p_DGazaNaVyhodeNagnetatelja.run ();
	END_IF;
END_IF
///////////////////////////////////////////////////
IF	kran3bOpen.start AND NOT kran3bOpen.top THEN//Проверяем, что открыт крана  3б
	IF	im.kran3b.onStatus=statusDualInput.STATUS_ON THEN
		kran3bOpen.top :=TRUE;	
	END_IF
END_IF
///////////////////////////////////////////////////
IF	kran3bOpen.top AND	kran5Close.top AND dP_kr1less100.top AND Pvh_vyhMore5.top THEN
	kran1Open.run ();  //кран 1 и 2 открываем
	kran2Open.run (); 
	kran3Open.run ();
	Smazka_1_2:=TRUE;
END_IF
IF	kran1Open.top THEN
	im.Kr_4_Open_From_Alg.off();
	ystavki.Block_kr4_alg.setValue (0);
END_IF
///////////////////////////////////////////////////
IF	kran1Open.top AND kran2Open.top AND kran3Open.top THEN //закрываем кран 3бис
	kran3bClose.run (); 
END_IF
///////////////////////////////////////////////////
IF 	kran3bClose.top THEN
	Err_ALG.error :=FALSE;
	timer480.reset ();
	end ();
ELSIF	(NOT (kran3bClose.top)) AND timer480.top THEN
		Err_ALG.error :=TRUE;
END_IF

METHOD PUBLIC reset
VAR_INPUT
END_VAR
SUPER^.reset();
im.Kr_4_Open_From_Alg.off();

statusSet.setBit(15,0);
END_METHOD

METHOD PUBLIC run
VAR_INPUT
END_VAR
SUPER^.run();
statusSet.setBit(15,1);
ystavki.Block_kr4_alg.setValue (1);
END_METHOD

END_FUNCTION_BLOCK

// K1/std12k5/Start_ALG/Kran_6_Close
{attribute 'symbol' := 'none'}
FUNCTION_BLOCK Kran_6_Close EXTENDS StepBySteapAlgoritm
VAR_INPUT
	
END_VAR
VAR_OUTPUT
	{attribute 'symbol' := 'read'}
	Kr_12_Move:		Question(table:=ADR(ObjectTable)):=			(AnswerVariants:=Answers.ANS_YES);
END_VAR
VAR
	K6_pusk:	ph_Kran (table:=ADR(phasesTable)):=			(phaseNumber:=0, Im:=Im.kran6, act:=DualStateImAction.off);
	K4_pusk:	ph_Kran (table:=ADR(phasesTable)):=			(phaseNumber:=1, Im:=Im.kran4, act:=DualStateImAction.off);
	timer5:		ph_Timer (table:=ADR(phasesTable)):=		(phaseNumber:=2, delay:=T#5S);
	Ypr_Kr1_2:	CustomPhase (table:=ADR(phasesTable)):=		(phaseNumber:=3);
END_VAR

SUPER^();
IF 	NOT K6_pusk.top THEN
	K6_pusk.run ();
END_IF
IF	K6_Pusk.top AND NOT K4_pusk.top THEN
	K4_pusk.run ();
END_IF

IF	K4_pusk.top THEN
	IF	((algmanager.mode = modegpa.MODE_PUSKAP_Ch) OR (algmanager.mode = modegpa.MODE_PUSKAP_R) OR (algmanager.mode = modegpa.MODE_PUSKPP_Ch) OR (algmanager.mode = modegpa.MODE_PUSKPP_R)) THEN
		timer5.run ();
		end();
	ELSE
		protections.p_kran1.run();
		protections.p_kran2.run();
		algoritms.Kr6_Move.canrun:=TRUE;
		algoritms.Kr6_Move.run();
		IF	im.PerepadDavlenieKran1_Less100.Q AND (algmanager.mode = modegpa.MODE_PUSKK) AND NOT Ypr_Kr1_2.top THEN
			Kr_12_Move.ask ();
		ELSE
			Kr_12_Move.reset ();
		END_IF
		IF	(Kr_12_Move.answer=Answers.ANS_YES) THEN
			
			Kr_12_Move.reset ();
			Ypr_Kr1_2.top:=TRUE;
		END_IF
		IF	Ypr_Kr1_2.top AND im.PerepadDavlenieKran1_Less100.Q THEN
			im.kran1.EnableOpcControl ();
			im.kran2.EnableOpcControl ();
		ELSE
			im.kran1.DisableOpcControl ();
			im.kran2.DisableOpcControl ();
		END_IF
		end();
	END_IF
END_IF

IF	timer5.top THEN
	algManager.setMode(nMode:=ModeGpa.MODE_WORK_M);
	algoritms.Kr6_Move.canrun:=TRUE;
	algoritms.Kr6_Move.run();
	protections.p_kran1.run();
	protections.p_kran2.run();
	reset ();
END_IF

METHOD PUBLIC reset
VAR_INPUT
END_VAR
SUPER^.reset();
im.kran1.DisableOpcControl ();
im.kran2.DisableOpcControl ();
Kr_12_Move.reset ();
END_METHOD

END_FUNCTION_BLOCK

// K2/std12k5/Start_ALG/Kran_6_Close
{attribute 'symbol' := 'none'}
FUNCTION_BLOCK Kran_6_Close EXTENDS StepBySteapAlgoritm
VAR_INPUT
	
END_VAR
VAR_OUTPUT
	{attribute 'symbol' := 'read'}
	Kr_12_Move:		Question(table:=ADR(ObjectTable)):=			(AnswerVariants:=Answers.ANS_YES);
END_VAR
VAR
	K6_pusk:	ph_Kran (table:=ADR(phasesTable)):=			(phaseNumber:=0, Im:=Im.kran6, act:=DualStateImAction.off);
	K4_pusk:	ph_Kran (table:=ADR(phasesTable)):=			(phaseNumber:=1, Im:=Im.kran4, act:=DualStateImAction.off);
	timer5:		ph_Timer (table:=ADR(phasesTable)):=		(phaseNumber:=2, delay:=T#5S);
	Ypr_Kr1_2:	CustomPhase (table:=ADR(phasesTable)):=		(phaseNumber:=3);
END_VAR

SUPER^();
IF 	NOT K6_pusk.top THEN
	K6_pusk.run ();
END_IF
IF	K6_Pusk.top AND NOT K4_pusk.top THEN
	K4_pusk.run ();
END_IF

IF	K4_pusk.top THEN
	IF	((algmanager.mode = modegpa.MODE_PUSKAP_Ch) OR (algmanager.mode = modegpa.MODE_PUSKAP_R) OR (algmanager.mode = modegpa.MODE_PUSKPP_Ch) OR (algmanager.mode = modegpa.MODE_PUSKPP_R)) THEN
		timer5.run ();
		end();
	ELSE
		protections.p_kran1.run();
		protections.p_kran2.run();
		algoritms.Kr6_Move.canrun:=TRUE;
		algoritms.Kr6_Move.run();
		IF	im.PerepadDavlenieKran1_Less100.Q AND (algmanager.mode = modegpa.MODE_PUSKK) AND NOT Ypr_Kr1_2.top THEN
			Kr_12_Move.ask ();
		ELSE
			Kr_12_Move.reset ();
		END_IF
		IF	(Kr_12_Move.answer=Answers.ANS_YES) THEN
			
			Kr_12_Move.reset ();
			Ypr_Kr1_2.top:=TRUE;
		END_IF
		IF	Ypr_Kr1_2.top AND im.PerepadDavlenieKran1_Less100.Q THEN
			im.kran1.EnableOpcControl ();
			im.kran2.EnableOpcControl ();
		ELSE
			im.kran1.DisableOpcControl ();
			im.kran2.DisableOpcControl ();
		END_IF
		end();
	END_IF
END_IF

IF	timer5.top THEN
	algManager.setMode(nMode:=ModeGpa.MODE_WORK_M);
	algoritms.Kr6_Move.canrun:=TRUE;
	algoritms.Kr6_Move.run();
	protections.p_kran1.run();
	protections.p_kran2.run();
	reset ();
END_IF

METHOD PUBLIC reset
VAR_INPUT
END_VAR
SUPER^.reset();
im.kran1.DisableOpcControl ();
im.kran2.DisableOpcControl ();
Kr_12_Move.reset ();
END_METHOD

END_FUNCTION_BLOCK

// K1/std12k5/Start_ALG/Kran_6_MOVE
{attribute 'symbol' := 'none'}
FUNCTION_BLOCK Kran_6_MOVE EXTENDS StepBySteapAlgoritm
VAR_INPUT
	
END_VAR
VAR_OUTPUT
	
END_VAR
VAR
	K6_pusk:	ph_Kran (table:=ADR(phasesTable)):=			(phaseNumber:=0, Im:=Im.kran6, act:=DualStateImAction.on);
	Kr6_Open:R_trig;
	Kr6_Close:R_trig;
END_VAR

SUPER^();
Kr6_Open (clk:= im.kran6.onStatus = statusDualInput.STATUS_On);
Kr6_Close (clk:= im.kran6.onStatus = statusDualInput.STATUS_Off);

IF	(algmanager.mode = modegpa.MODE_WORK_M) AND Kr6_Open.Q THEN
	algManager.setMode(nMode:=ModeGpa.MODE_WORK_K);
END_IF
IF	(algmanager.mode = modegpa.MODE_WORK_K) AND Kr6_Close.Q THEN
	algManager.setMode(nMode:=ModeGpa.MODE_WORK_M);
END_IF


IF (algmanager.mode = modegpa.MODE_WORK_M) AND (ai.TokStatora.interval >= statusAi.NORMAL) AND (ai.TokStatora.value <= 240 ) THEN
	K6_pusk.run ();
	im.kran6.DisableOpcControl();
END_IF
IF	(K6_pusk.top AND (ai.TokStatora.interval >= statusAi.NORMAL) AND (ai.TokStatora.value > 240)) THEN
	K6_pusk.reset ();
	im.kran6.EnableOpcControl();
END_IF

IF (algmanager.mode = modegpa.MODE_WORK_M) THEN
	algoritms.S_Vibr.CanRun:=TRUE;
	algoritms.S_Vibr.run ();
ELSE
	algoritms.S_Vibr.CanRun:=FALSE;
	algoritms.S_Vibr.reset ();
END_IF

METHOD PUBLIC reset
VAR_INPUT
END_VAR
SUPER^.reset();
im.kran6.DisableOpcControl();
im.kran1.DisableOpcControl	 ();
im.kran2.DisableOpcControl ();
END_METHOD

METHOD PUBLIC run
VAR_INPUT
END_VAR
SUPER^.run();
im.kran6.EnableOpcControl();
END_METHOD

END_FUNCTION_BLOCK

// K2/std12k5/Start_ALG/Kran_6_MOVE
{attribute 'symbol' := 'none'}
FUNCTION_BLOCK Kran_6_MOVE EXTENDS StepBySteapAlgoritm
VAR_INPUT
	
END_VAR
VAR_OUTPUT
	
END_VAR
VAR
	K6_pusk:	ph_Kran (table:=ADR(phasesTable)):=			(phaseNumber:=0, Im:=Im.kran6, act:=DualStateImAction.on);
	Kr6_Open:R_trig;
	Kr6_Close:R_trig;
END_VAR

SUPER^();
Kr6_Open (clk:= im.kran6.onStatus = statusDualInput.STATUS_On);
Kr6_Close (clk:= im.kran6.onStatus = statusDualInput.STATUS_Off);

IF	(algmanager.mode = modegpa.MODE_WORK_M) AND Kr6_Open.Q THEN
	algManager.setMode(nMode:=ModeGpa.MODE_WORK_K);
END_IF
IF	(algmanager.mode = modegpa.MODE_WORK_K) AND Kr6_Close.Q THEN
	algManager.setMode(nMode:=ModeGpa.MODE_WORK_M);
END_IF


IF (algmanager.mode = modegpa.MODE_WORK_M) AND (ai.TokStatora.interval >= statusAi.NORMAL) AND (ai.TokStatora.value <= 240 ) THEN
	K6_pusk.run ();
	im.kran6.DisableOpcControl();
END_IF
IF	(K6_pusk.top AND (ai.TokStatora.interval >= statusAi.NORMAL) AND (ai.TokStatora.value > 240)) THEN
	K6_pusk.reset ();
	im.kran6.EnableOpcControl();
END_IF

IF (algmanager.mode = modegpa.MODE_WORK_M) THEN
	algoritms.S_Vibr.CanRun:=TRUE;
	algoritms.S_Vibr.run ();
ELSE
	algoritms.S_Vibr.CanRun:=FALSE;
	algoritms.S_Vibr.reset ();
END_IF

METHOD PUBLIC reset
VAR_INPUT
END_VAR
SUPER^.reset();
im.kran6.DisableOpcControl();
im.kran1.DisableOpcControl	 ();
im.kran2.DisableOpcControl ();
END_METHOD

METHOD PUBLIC run
VAR_INPUT
END_VAR
SUPER^.run();
im.kran6.EnableOpcControl();
END_METHOD

END_FUNCTION_BLOCK

// K1/std12k5/Start_ALG/PNS_Pusk
{attribute 'symbol' := 'none'}
FUNCTION_BLOCK PNS_Pusk EXTENDS StepBySteapAlgoritm
VAR_INPUT
	
END_VAR
VAR_OUTPUT
	{attribute 'symbol' := 'read'}
	AutoPNS_Ask:		Question(table:=ADR(ObjectTable)):=			(AnswerVariants:=Answers.ANS_YES);
END_VAR
VAR
	{attribute 'symbol' := 'read'}
	timer600:		ph_Timer (table:=ADR(phasesTable)):=		(phaseNumber:=0, delay:=T#600S);
	pnsOff:			ph_Switch 	(table:=ADR(phasesTable)):=		(phaseNumber:=1, Im:=Im.pns, act:=DualStateImAction.off);
	StartAutoPNS:	ph_algoritm (table:=ADR(phasesTable)):=		(phaseNumber:=2, Im:=algoritms.autoPns, act:=PhaseAlgoritmAction.run,waitCompletion:=FALSE);
	timer5:			ph_Timer (table:=ADR(phasesTable)):=		(phaseNumber:=3, delay:=T#5S);
	PNS_Off_cmd:	CustomPhase (table:=ADR(phasesTable)):=		(phaseNumber:=4);
END_VAR

SUPER^();

IF	(NOT (AutoPNS_Ask.answer=Answers.ANS_YES)) AND (NOT timer600.top) AND ((algmanager.mode = modegpa.MODE_PUSKAP_R) OR (algmanager.mode = modegpa.MODE_PUSKPP_R)
	OR (algmanager.mode = modegpa.MODE_PUSKAP_Ch) OR (algmanager.mode = modegpa.MODE_PUSKPP_Ch)) AND NOT StartAutoPNS.start AND NOT PNS_Off_cmd.top THEN
	timer600.run ();
END_IF;

IF	(NOT timer600.top) AND NOT StartAutoPNS.start AND NOT PNS_Off_cmd.top THEN
	AutoPNS_Ask.ask();
END_IF


IF	(timer600.top) OR (AutoPNS_Ask.answer=Answers.ANS_YES) THEN
	AutoPNS_Ask.reset ();
	pnsOff.run ();
	timer600.reset ();	
	PNS_Off_cmd.top:=TRUE;
END_IF
IF	PNS_Off_cmd.top AND pnsOff.top THEN
	algoritms.autoPns.CanRun:=TRUE;
	StartAutoPNS.run ();
END_IF
IF	StartAutoPNS.top THEN
	timer5.run ();
	end ();
END_IF
IF	timer5.top THEN
	timer5.reset ();
	reset ();
END_IF;

METHOD PUBLIC reset
VAR_INPUT
END_VAR
SUPER^.reset();
AutoPNS_Ask.reset ();
END_METHOD

END_FUNCTION_BLOCK

// K2/std12k5/Start_ALG/PNS_Pusk
{attribute 'symbol' := 'none'}
FUNCTION_BLOCK PNS_Pusk EXTENDS StepBySteapAlgoritm
VAR_INPUT
	
END_VAR
VAR_OUTPUT
	{attribute 'symbol' := 'read'}
	AutoPNS_Ask:		Question(table:=ADR(ObjectTable)):=			(AnswerVariants:=Answers.ANS_YES);
END_VAR
VAR
	{attribute 'symbol' := 'read'}
	timer600:		ph_Timer (table:=ADR(phasesTable)):=		(phaseNumber:=0, delay:=T#600S);
	pnsOff:			ph_Switch 	(table:=ADR(phasesTable)):=		(phaseNumber:=1, Im:=Im.pns, act:=DualStateImAction.off);
	StartAutoPNS:	ph_algoritm (table:=ADR(phasesTable)):=		(phaseNumber:=2, Im:=algoritms.autoPns, act:=PhaseAlgoritmAction.run,waitCompletion:=FALSE);
	timer5:			ph_Timer (table:=ADR(phasesTable)):=		(phaseNumber:=3, delay:=T#5S);
	PNS_Off_cmd:	CustomPhase (table:=ADR(phasesTable)):=		(phaseNumber:=4);
END_VAR

SUPER^();

IF	(NOT (AutoPNS_Ask.answer=Answers.ANS_YES)) AND (NOT timer600.top) AND ((algmanager.mode = modegpa.MODE_PUSKAP_R) OR (algmanager.mode = modegpa.MODE_PUSKPP_R)
	OR (algmanager.mode = modegpa.MODE_PUSKAP_Ch) OR (algmanager.mode = modegpa.MODE_PUSKPP_Ch)) AND NOT StartAutoPNS.start AND NOT PNS_Off_cmd.top THEN
	timer600.run ();
END_IF;

IF	(NOT timer600.top) AND NOT StartAutoPNS.start AND NOT PNS_Off_cmd.top THEN
	AutoPNS_Ask.ask();
END_IF


IF	(timer600.top) OR (AutoPNS_Ask.answer=Answers.ANS_YES) THEN
	AutoPNS_Ask.reset ();
	pnsOff.run ();
	timer600.reset ();	
	PNS_Off_cmd.top:=TRUE;
END_IF
IF	PNS_Off_cmd.top AND pnsOff.top THEN
	algoritms.autoPns.CanRun:=TRUE;
	StartAutoPNS.run ();
END_IF
IF	StartAutoPNS.top THEN
	timer5.run ();
	end ();
END_IF
IF	timer5.top THEN
	timer5.reset ();
	reset ();
END_IF;

METHOD PUBLIC reset
VAR_INPUT
END_VAR
SUPER^.reset();
AutoPNS_Ask.reset ();
END_METHOD

END_FUNCTION_BLOCK

// K1/std12k5/Start_ALG/Reset_AutoAVOM
{attribute 'symbol' := 'none'}
FUNCTION_BLOCK Reset_AutoAVOM EXTENDS StepBySteapAlgoritm
VAR_INPUT
END_VAR
	
VAR_OUTPUT
	{attribute 'symbol' := 'read'}
	Start_Prov_Pusk:		Question(table:=ADR(ObjectTable)):=			(AnswerVariants:=(Answers.ANS_YES OR Answers.ANS_NO));
END_VAR
VAR
	Alg_Start_reset:	ph_algoritm (table:=ADR(phasesTable)):=		(phaseNumber:=0, Im:=algoritms.Auto_Avom_ , act:=PhaseAlgoritmAction.reset, waitCompletion:=FALSE);
END_VAR

SUPER^();
IF	NOT Alg_Start_reset.start THEN
	Start_Prov_Pusk.ask ();
END_IF
IF	(Start_Prov_Pusk.answer=Answers.ANS_YES) THEN
	algoritms.Auto_Avom_.CanRun:=FALSE;
	Alg_Start_reset.run ();
	Start_Prov_Pusk.reset ();
	reset ();
ELSIF	(Start_Prov_Pusk.answer=Answers.ANS_NO) THEN
		Start_Prov_Pusk.reset ();
		algoritms.Auto_Avom_.CanRun:=TRUE;
		reset ();
		
END_IF

METHOD PUBLIC reset
VAR_INPUT
END_VAR
SUPER^.reset();
Start_Prov_Pusk.reset ();
END_METHOD

END_FUNCTION_BLOCK

// K2/std12k5/Start_ALG/Reset_AutoAVOM
{attribute 'symbol' := 'none'}
FUNCTION_BLOCK Reset_AutoAVOM EXTENDS StepBySteapAlgoritm
VAR_INPUT
END_VAR
	
VAR_OUTPUT
	{attribute 'symbol' := 'read'}
	Start_Prov_Pusk:		Question(table:=ADR(ObjectTable)):=			(AnswerVariants:=(Answers.ANS_YES OR Answers.ANS_NO));
END_VAR
VAR
	Alg_Start_reset:	ph_algoritm (table:=ADR(phasesTable)):=		(phaseNumber:=0, Im:=algoritms.Auto_Avom_ , act:=PhaseAlgoritmAction.reset, waitCompletion:=FALSE);
END_VAR

SUPER^();
IF	NOT Alg_Start_reset.start THEN
	Start_Prov_Pusk.ask ();
END_IF
IF	(Start_Prov_Pusk.answer=Answers.ANS_YES) THEN
	algoritms.Auto_Avom_.CanRun:=FALSE;
	Alg_Start_reset.run ();
	Start_Prov_Pusk.reset ();
	reset ();
ELSIF	(Start_Prov_Pusk.answer=Answers.ANS_NO) THEN
		Start_Prov_Pusk.reset ();
		algoritms.Auto_Avom_.CanRun:=TRUE;
		reset ();
		
END_IF

METHOD PUBLIC reset
VAR_INPUT
END_VAR
SUPER^.reset();
Start_Prov_Pusk.reset ();
END_METHOD

END_FUNCTION_BLOCK

// K1/std12k5/Start_ALG/Reset_AutoTEN
{attribute 'symbol' := 'none'}
FUNCTION_BLOCK Reset_AutoTEN EXTENDS StepBySteapAlgoritm
VAR_INPUT
END_VAR
	
VAR_OUTPUT
	{attribute 'symbol' := 'read'}
	Start_Prov_Pusk:		Question(table:=ADR(ObjectTable)):=			(AnswerVariants:=(Answers.ANS_YES OR Answers.ANS_NO));
END_VAR
VAR
	Alg_Start_reset:	ph_algoritm (table:=ADR(phasesTable)):=		(phaseNumber:=0, Im:=algoritms.AUto_Ten_ , act:=PhaseAlgoritmAction.reset, waitCompletion:=FALSE);
END_VAR

SUPER^();
IF	NOT Alg_Start_reset.start THEN
	Start_Prov_Pusk.ask ();
END_IF
IF	(Start_Prov_Pusk.answer=Answers.ANS_YES) THEN
	algoritms.AUto_Ten_.CanRun:=FALSE;
	Alg_Start_reset.run ();
	Start_Prov_Pusk.reset ();
	reset ();
ELSIF	(Start_Prov_Pusk.answer=Answers.ANS_NO) THEN
		algoritms.AUto_Ten_.CanRun:=TRUE;
		Start_Prov_Pusk.reset ();
		reset ();
		
END_IF

METHOD PUBLIC reset
VAR_INPUT
END_VAR
SUPER^.reset();
Start_Prov_Pusk.reset ();
END_METHOD

END_FUNCTION_BLOCK

// K2/std12k5/Start_ALG/Reset_AutoTEN
{attribute 'symbol' := 'none'}
FUNCTION_BLOCK Reset_AutoTEN EXTENDS StepBySteapAlgoritm
VAR_INPUT
END_VAR
	
VAR_OUTPUT
	{attribute 'symbol' := 'read'}
	Start_Prov_Pusk:		Question(table:=ADR(ObjectTable)):=			(AnswerVariants:=(Answers.ANS_YES OR Answers.ANS_NO));
END_VAR
VAR
	Alg_Start_reset:	ph_algoritm (table:=ADR(phasesTable)):=		(phaseNumber:=0, Im:=algoritms.AUto_Ten_ , act:=PhaseAlgoritmAction.reset, waitCompletion:=FALSE);
END_VAR

SUPER^();
IF	NOT Alg_Start_reset.start THEN
	Start_Prov_Pusk.ask ();
END_IF
IF	(Start_Prov_Pusk.answer=Answers.ANS_YES) THEN
	algoritms.AUto_Ten_.CanRun:=FALSE;
	Alg_Start_reset.run ();
	Start_Prov_Pusk.reset ();
	reset ();
ELSIF	(Start_Prov_Pusk.answer=Answers.ANS_NO) THEN
		algoritms.AUto_Ten_.CanRun:=TRUE;
		Start_Prov_Pusk.reset ();
		reset ();
		
END_IF

METHOD PUBLIC reset
VAR_INPUT
END_VAR
SUPER^.reset();
Start_Prov_Pusk.reset ();
END_METHOD

END_FUNCTION_BLOCK

// K1/std12k5/Start_ALG/Reset_Test_IM
{attribute 'symbol' := 'none'}
FUNCTION_BLOCK Reset_Test_IM EXTENDS StepBySteapAlgoritm
VAR_INPUT
END_VAR
	
VAR_OUTPUT
	{attribute 'symbol' := 'read'}
	Start_Prov_Pusk:		Question(table:=ADR(ObjectTable)):=			(AnswerVariants:=(Answers.ANS_YES OR Answers.ANS_NO));
END_VAR
VAR
	Alg_Start_reset:	ph_algoritm (table:=ADR(phasesTable)):=		(phaseNumber:=0, Im:=algoritms.Test_IM, act:=PhaseAlgoritmAction.reset, waitCompletion:=FALSE);
END_VAR

SUPER^();
IF	NOT Alg_Start_reset.start THEN
	Start_Prov_Pusk.ask ();
END_IF
IF	(Start_Prov_Pusk.answer=Answers.ANS_YES) THEN
	algoritms.Test_IM.CanRun:=FALSE;
	Alg_Start_reset.run ();
	Start_Prov_Pusk.reset ();
	reset ();
ELSIF	(Start_Prov_Pusk.answer=Answers.ANS_NO) THEN
		IF	algoritms.Test_IM.isRuning THEN
			algoritms.Test_IM.CanRun:=TRUE;
			Start_Prov_Pusk.reset ();
			reset ();
		ELSIF	NOT algoritms.Test_IM.CanRun THEN
			Start_Prov_Pusk.reset ();
			reset ();
		END_IF	
END_IF

METHOD PUBLIC reset
VAR_INPUT
END_VAR
SUPER^.reset();
Start_Prov_Pusk.reset ();
END_METHOD

END_FUNCTION_BLOCK

// K2/std12k5/Start_ALG/Reset_Test_IM
{attribute 'symbol' := 'none'}
FUNCTION_BLOCK Reset_Test_IM EXTENDS StepBySteapAlgoritm
VAR_INPUT
END_VAR
	
VAR_OUTPUT
	{attribute 'symbol' := 'read'}
	Start_Prov_Pusk:		Question(table:=ADR(ObjectTable)):=			(AnswerVariants:=(Answers.ANS_YES OR Answers.ANS_NO));
END_VAR
VAR
	Alg_Start_reset:	ph_algoritm (table:=ADR(phasesTable)):=		(phaseNumber:=0, Im:=algoritms.Test_IM, act:=PhaseAlgoritmAction.reset, waitCompletion:=FALSE);
END_VAR

SUPER^();
IF	NOT Alg_Start_reset.start THEN
	Start_Prov_Pusk.ask ();
END_IF
IF	(Start_Prov_Pusk.answer=Answers.ANS_YES) THEN
	algoritms.Test_IM.CanRun:=FALSE;
	Alg_Start_reset.run ();
	Start_Prov_Pusk.reset ();
	reset ();
ELSIF	(Start_Prov_Pusk.answer=Answers.ANS_NO) THEN
		IF	algoritms.Test_IM.isRuning THEN
			algoritms.Test_IM.CanRun:=TRUE;
			Start_Prov_Pusk.reset ();
			reset ();
		ELSIF	NOT algoritms.Test_IM.CanRun THEN
			Start_Prov_Pusk.reset ();
			reset ();
		END_IF	
END_IF

METHOD PUBLIC reset
VAR_INPUT
END_VAR
SUPER^.reset();
Start_Prov_Pusk.reset ();
END_METHOD

END_FUNCTION_BLOCK

// K1/std12k5/Start_ALG/Start_AutoAVOM
{attribute 'symbol' := 'none'}
FUNCTION_BLOCK Start_AutoAVOM EXTENDS StepBySteapAlgoritm
VAR_INPUT
END_VAR
	
VAR_OUTPUT
	{attribute 'symbol' := 'read'}
	Start_Prov_Pusk:		Question(table:=ADR(ObjectTable)):=			(AnswerVariants:=(Answers.ANS_YES OR Answers.ANS_NO));
END_VAR
VAR
	Alg_Start_reset:	ph_algoritm (table:=ADR(phasesTable)):=		(phaseNumber:=0, Im:=algoritms.Auto_Avom_, act:=PhaseAlgoritmAction.run, waitCompletion:=FALSE);
END_VAR

SUPER^();
IF 	NOT Alg_Start_reset.start AND ((Ystavki.num_avom.Yst [0] <> Ystavki.num_avom.Yst [1]) AND  (Ystavki.num_avom.Yst [0] <> Ystavki.num_avom.Yst [2]) AND  (Ystavki.num_avom.Yst [0] <> Ystavki.num_avom.Yst [3]) AND
	(Ystavki.num_avom.Yst [1] <> Ystavki.num_avom.Yst [2]) AND (Ystavki.num_avom.Yst [1] <> Ystavki.num_avom.Yst [3]) AND (Ystavki.num_avom.Yst [2] <> Ystavki.num_avom.Yst [3]) AND (Ystavki.num_avom.Yst [0] >= 1) AND (Ystavki.num_avom.Yst [0] <= 4) 
	AND (Ystavki.num_avom.Yst [1] >= 1) AND (Ystavki.num_avom.Yst [1] <= 4) AND (Ystavki.num_avom.Yst [2] >= 1) AND (Ystavki.num_avom.Yst [2] <= 4)	AND (Ystavki.num_avom.Yst [3] >= 1) AND (Ystavki.num_avom.Yst [3] <= 4)) THEN
	Start_Prov_Pusk.ask ();
ELSE
	Start_Prov_Pusk.reset ();
	algoritms.Auto_AVOM_.CanRun:=FALSE;
	reset ();
end_if;
IF	(Start_Prov_Pusk.answer=Answers.ANS_YES)  THEN
	algoritms.Auto_Avom_.CanRun:=TRUE;
	Alg_Start_reset.run ();
	Start_Prov_Pusk.reset ();
	reset ();
ELSIF	(Start_Prov_Pusk.answer=Answers.ANS_NO) THEN
		Start_Prov_Pusk.reset ();
		algoritms.Auto_AVOM_.CanRun:=FALSE;
		reset ();
END_IF

METHOD PUBLIC reset
VAR_INPUT
END_VAR
SUPER^.reset();
Start_Prov_Pusk.reset ();
END_METHOD

END_FUNCTION_BLOCK

// K2/std12k5/Start_ALG/Start_AutoAVOM
{attribute 'symbol' := 'none'}
FUNCTION_BLOCK Start_AutoAVOM EXTENDS StepBySteapAlgoritm
VAR_INPUT
END_VAR
	
VAR_OUTPUT
	{attribute 'symbol' := 'read'}
	Start_Prov_Pusk:		Question(table:=ADR(ObjectTable)):=			(AnswerVariants:=(Answers.ANS_YES OR Answers.ANS_NO));
END_VAR
VAR
	Alg_Start_reset:	ph_algoritm (table:=ADR(phasesTable)):=		(phaseNumber:=0, Im:=algoritms.Auto_Avom_, act:=PhaseAlgoritmAction.run, waitCompletion:=FALSE);
END_VAR

SUPER^();
IF 	NOT Alg_Start_reset.start AND ((Ystavki.num_avom.Yst [0] <> Ystavki.num_avom.Yst [1]) AND  (Ystavki.num_avom.Yst [0] <> Ystavki.num_avom.Yst [2]) AND  (Ystavki.num_avom.Yst [0] <> Ystavki.num_avom.Yst [3]) AND
	(Ystavki.num_avom.Yst [1] <> Ystavki.num_avom.Yst [2]) AND (Ystavki.num_avom.Yst [1] <> Ystavki.num_avom.Yst [3]) AND (Ystavki.num_avom.Yst [2] <> Ystavki.num_avom.Yst [3]) AND (Ystavki.num_avom.Yst [0] >= 1) AND (Ystavki.num_avom.Yst [0] <= 4) 
	AND (Ystavki.num_avom.Yst [1] >= 1) AND (Ystavki.num_avom.Yst [1] <= 4) AND (Ystavki.num_avom.Yst [2] >= 1) AND (Ystavki.num_avom.Yst [2] <= 4)	AND (Ystavki.num_avom.Yst [3] >= 1) AND (Ystavki.num_avom.Yst [3] <= 4)) THEN
	Start_Prov_Pusk.ask ();
ELSE
	Start_Prov_Pusk.reset ();
	algoritms.Auto_AVOM_.CanRun:=FALSE;
	reset ();
end_if;
IF	(Start_Prov_Pusk.answer=Answers.ANS_YES)  THEN
	algoritms.Auto_Avom_.CanRun:=TRUE;
	Alg_Start_reset.run ();
	Start_Prov_Pusk.reset ();
	reset ();
ELSIF	(Start_Prov_Pusk.answer=Answers.ANS_NO) THEN
		Start_Prov_Pusk.reset ();
		algoritms.Auto_AVOM_.CanRun:=FALSE;
		reset ();
END_IF

METHOD PUBLIC reset
VAR_INPUT
END_VAR
SUPER^.reset();
Start_Prov_Pusk.reset ();
END_METHOD

END_FUNCTION_BLOCK

// K1/std12k5/Start_ALG/Start_AutoTEN
{attribute 'symbol' := 'none'}
FUNCTION_BLOCK Start_AutoTEN EXTENDS StepBySteapAlgoritm
VAR_INPUT
END_VAR
	
VAR_OUTPUT
	{attribute 'symbol' := 'read'}
	Start_Prov_Pusk:		Question(table:=ADR(ObjectTable)):=			(AnswerVariants:=(Answers.ANS_YES OR Answers.ANS_NO));
END_VAR
VAR
	Alg_Start_reset:	ph_algoritm (table:=ADR(phasesTable)):=		(phaseNumber:=0, Im:=algoritms.AUto_Ten_, act:=PhaseAlgoritmAction.run, waitCompletion:=FALSE);
END_VAR

SUPER^();
IF	NOT Alg_Start_reset.start THEN
	Start_Prov_Pusk.ask ();
END_IF
IF	(Start_Prov_Pusk.answer=Answers.ANS_YES) THEN
	algoritms.AUto_Ten_.CanRun:=TRUE;
	Alg_Start_reset.run ();
	Start_Prov_Pusk.reset ();
	reset ();
ELSIF	(Start_Prov_Pusk.answer=Answers.ANS_NO) THEN
		algoritms.AUto_Ten_.CanRun:=FALSE;
		Start_Prov_Pusk.reset ();
		reset ();
END_IF

METHOD PUBLIC reset
VAR_INPUT
END_VAR
SUPER^.reset();
Start_Prov_Pusk.reset ();
END_METHOD

END_FUNCTION_BLOCK

// K2/std12k5/Start_ALG/Start_AutoTEN
{attribute 'symbol' := 'none'}
FUNCTION_BLOCK Start_AutoTEN EXTENDS StepBySteapAlgoritm
VAR_INPUT
END_VAR
	
VAR_OUTPUT
	{attribute 'symbol' := 'read'}
	Start_Prov_Pusk:		Question(table:=ADR(ObjectTable)):=			(AnswerVariants:=(Answers.ANS_YES OR Answers.ANS_NO));
END_VAR
VAR
	Alg_Start_reset:	ph_algoritm (table:=ADR(phasesTable)):=		(phaseNumber:=0, Im:=algoritms.AUto_Ten_, act:=PhaseAlgoritmAction.run, waitCompletion:=FALSE);
END_VAR

SUPER^();
IF	NOT Alg_Start_reset.start THEN
	Start_Prov_Pusk.ask ();
END_IF
IF	(Start_Prov_Pusk.answer=Answers.ANS_YES) THEN
	algoritms.AUto_Ten_.CanRun:=TRUE;
	Alg_Start_reset.run ();
	Start_Prov_Pusk.reset ();
	reset ();
ELSIF	(Start_Prov_Pusk.answer=Answers.ANS_NO) THEN
		algoritms.AUto_Ten_.CanRun:=FALSE;
		Start_Prov_Pusk.reset ();
		reset ();
END_IF

METHOD PUBLIC reset
VAR_INPUT
END_VAR
SUPER^.reset();
Start_Prov_Pusk.reset ();
END_METHOD

END_FUNCTION_BLOCK

// K1/std12k5/Start_ALG/Start_ProtectionsVibr
{attribute 'symbol' := 'none'}
FUNCTION_BLOCK Start_ProtectionsVibr EXTENDS StepBySteapAlgoritm
VAR_INPUT
END_VAR
VAR_OUTPUT
END_VAR
VAR
	{attribute 'symbol' := 'read'}
	timer20:	ph_Timer 	(table:=ADR(phasesTable)):=		(phaseNumber:=0, delay:=T#20S);
END_VAR

SUPER^();
IF	NOT timer20.top THEN
	timer20.run ();
END_IF

IF	timer20.top THEN
	protections.p_VibroSkorostOPED_T1.run ();
	protections.p_VibroSkorostOPShesterniReduktoraH_T6.run ();
	protections.p_VibroSkorostOYPED_T2.run ();
	protections.p_VibroSkorostOYPKolesaED_T3.run ();
	protections.p_VibroSkorostOPKolesaRH_T4.run ();
	protections.p_VibroSkorostOPShesterniRED_T5.run ();
	end();
END_IF

METHOD PUBLIC reset
VAR_INPUT
END_VAR
SUPER^.reset();
protections.p_VibroSkorostOPED_T1.reset ();
protections.p_VibroSkorostOPShesterniReduktoraH_T6.reset ();
protections.p_VibroSkorostOYPED_T2.reset ();
protections.p_VibroSkorostOYPKolesaED_T3.reset ();
protections.p_VibroSkorostOPKolesaRH_T4.reset ();
protections.p_VibroSkorostOPShesterniRED_T5.reset  ();
timer20.reset ();
END_METHOD

END_FUNCTION_BLOCK

// K2/std12k5/Start_ALG/Start_ProtectionsVibr
{attribute 'symbol' := 'none'}
FUNCTION_BLOCK Start_ProtectionsVibr EXTENDS StepBySteapAlgoritm
VAR_INPUT
END_VAR
VAR_OUTPUT
END_VAR
VAR
	{attribute 'symbol' := 'read'}
	timer20:	ph_Timer 	(table:=ADR(phasesTable)):=		(phaseNumber:=0, delay:=T#20S);
END_VAR

SUPER^();
IF	NOT timer20.top THEN
	timer20.run ();
END_IF

IF	timer20.top THEN
	protections.p_VibroSkorostOPED_T1.run ();
	protections.p_VibroSkorostOPShesterniReduktoraH_T6.run ();
	protections.p_VibroSkorostOYPED_T2.run ();
	protections.p_VibroSkorostOYPKolesaED_T3.run ();
	protections.p_VibroSkorostOPKolesaRH_T4.run ();
	protections.p_VibroSkorostOPShesterniRED_T5.run ();
	end();
END_IF

METHOD PUBLIC reset
VAR_INPUT
END_VAR
SUPER^.reset();
protections.p_VibroSkorostOPED_T1.reset ();
protections.p_VibroSkorostOPShesterniReduktoraH_T6.reset ();
protections.p_VibroSkorostOYPED_T2.reset ();
protections.p_VibroSkorostOYPKolesaED_T3.reset ();
protections.p_VibroSkorostOPKolesaRH_T4.reset ();
protections.p_VibroSkorostOPShesterniRED_T5.reset  ();
timer20.reset ();
END_METHOD

END_FUNCTION_BLOCK

// K1/std12k5/Start_ALG/Start_Prov_dPmg
{attribute 'symbol' := 'none'}
FUNCTION_BLOCK Start_Prov_dPmg EXTENDS StepBySteapAlgoritm
VAR_INPUT
END_VAR
VAR_OUTPUT
	{attribute 'symbol' := 'read'}
	Start_Prov_Pusk:		Question(table:=ADR(ObjectTable)):=			(AnswerVariants:=(Answers.ANS_YES OR Answers.ANS_NO));
END_VAR
VAR
	F1_1_start:		ph_algoritm (table:=ADR(phasesTable)):=		(phaseNumber:=0, Im:=algoritms.F1_1, act:=PhaseAlgoritmAction.run, waitCompletion:=TRUE);
	F1_2_start: 	ph_algoritm (table:=ADR(phasesTable)):=	(phaseNumber:=1, Im:=algoritms.F1_2, act:=PhaseAlgoritmAction.run, waitCompletion:=TRUE);
	dPmg_start: 	ph_algoritm (table:=ADR(phasesTable)):=	(phaseNumber:=2, Im:=algoritms.dPmg, act:=PhaseAlgoritmAction.run, waitCompletion:=TRUE);
END_VAR

SUPER^();
IF	NOT F1_1_start.start THEN
	Start_Prov_Pusk.ask ();
END_IF
IF	(Start_Prov_Pusk.answer=Answers.ANS_YES) THEN
	algManager.setMode(nMode:=ModeGpa.MODE_PROBDPMG);
	algoritms.F1_1.CanRun:=TRUE;
	F1_1_start.run ();
	Start_Prov_Pusk.reset ();
ELSIF	(Start_Prov_Pusk.answer=Answers.ANS_NO) THEN
		Start_Prov_Pusk.reset ();
		algoritms.F1_1.CanRun:=FALSE;
		reset ();
END_IF


IF 	F1_1_start.top THEN
	algoritms.F1_2.CanRun:=TRUE;
	F1_2_start.run ();
END_IF
IF 	F1_2_start.top THEN
	algoritms.dPmg.CanRun:=TRUE;
	dPmg_start.run ();
	reset ();
END_IF

METHOD PUBLIC reset
VAR_INPUT
END_VAR
SUPER^.reset();
Start_Prov_Pusk.reset ();
END_METHOD

END_FUNCTION_BLOCK

// K2/std12k5/Start_ALG/Start_Prov_dPmg
{attribute 'symbol' := 'none'}
FUNCTION_BLOCK Start_Prov_dPmg EXTENDS StepBySteapAlgoritm
VAR_INPUT
END_VAR
VAR_OUTPUT
	{attribute 'symbol' := 'read'}
	Start_Prov_Pusk:		Question(table:=ADR(ObjectTable)):=			(AnswerVariants:=(Answers.ANS_YES OR Answers.ANS_NO));
END_VAR
VAR
	F1_1_start:		ph_algoritm (table:=ADR(phasesTable)):=		(phaseNumber:=0, Im:=algoritms.F1_1, act:=PhaseAlgoritmAction.run, waitCompletion:=TRUE);
	F1_2_start: 	ph_algoritm (table:=ADR(phasesTable)):=	(phaseNumber:=1, Im:=algoritms.F1_2, act:=PhaseAlgoritmAction.run, waitCompletion:=TRUE);
	dPmg_start: 	ph_algoritm (table:=ADR(phasesTable)):=	(phaseNumber:=2, Im:=algoritms.dPmg, act:=PhaseAlgoritmAction.run, waitCompletion:=TRUE);
END_VAR

SUPER^();
IF	NOT F1_1_start.start THEN
	Start_Prov_Pusk.ask ();
END_IF
IF	(Start_Prov_Pusk.answer=Answers.ANS_YES) THEN
	algManager.setMode(nMode:=ModeGpa.MODE_PROBDPMG);
	algoritms.F1_1.CanRun:=TRUE;
	F1_1_start.run ();
	Start_Prov_Pusk.reset ();
ELSIF	(Start_Prov_Pusk.answer=Answers.ANS_NO) THEN
		Start_Prov_Pusk.reset ();
		algoritms.F1_1.CanRun:=FALSE;
		reset ();
END_IF


IF 	F1_1_start.top THEN
	algoritms.F1_2.CanRun:=TRUE;
	F1_2_start.run ();
END_IF
IF 	F1_2_start.top THEN
	algoritms.dPmg.CanRun:=TRUE;
	dPmg_start.run ();
	reset ();
END_IF

METHOD PUBLIC reset
VAR_INPUT
END_VAR
SUPER^.reset();
Start_Prov_Pusk.reset ();
END_METHOD

END_FUNCTION_BLOCK

// K1/std12k5/Start_ALG/Start_Prov_I
{attribute 'symbol' := 'none'}
FUNCTION_BLOCK Start_Prov_I EXTENDS StepBySteapAlgoritm
VAR_INPUT
END_VAR
VAR_OUTPUT
	{attribute 'symbol' := 'read'}
	Start_Prov_Pusk:		Question(table:=ADR(ObjectTable)):=			(AnswerVariants:=(Answers.ANS_YES OR Answers.ANS_NO));
	{attribute 'symbol' := 'read'}
	F4_Start_Q:		Question(table:=ADR(ObjectTable)):=			(AnswerVariants:=Answers.ANS_YES);
END_VAR
VAR
	F1_1_start:	ph_algoritm (table:=ADR(phasesTable)):=		(phaseNumber:=0, Im:=algoritms.F1_1 , act:=PhaseAlgoritmAction.run, waitCompletion:=TRUE);
	F1_2_start:	ph_algoritm (table:=ADR(phasesTable)):=		(phaseNumber:=1, Im:=algoritms.F1_2 , act:=PhaseAlgoritmAction.run, waitCompletion:=TRUE);
	F2_Start: ph_algoritm (table:=ADR(phasesTable)):=		(phaseNumber:=2, Im:=algoritms.F2_R , act:=PhaseAlgoritmAction.run, waitCompletion:=TRUE);
	F3_Start: ph_algoritm (table:=ADR(phasesTable)):=		(phaseNumber:=3, Im:=algoritms.F3 , act:=PhaseAlgoritmAction.run, waitCompletion:=TRUE);
	F4_Start: ph_algoritm (table:=ADR(phasesTable)):=		(phaseNumber:=4, Im:=algoritms.F4 , act:=PhaseAlgoritmAction.run, waitCompletion:=TRUE);
END_VAR

SUPER^();
IF	NOT F1_1_start.start THEN
	Start_Prov_Pusk.ask ();
END_IF
IF	(Start_Prov_Pusk.answer=Answers.ANS_YES) THEN
	algManager.setMode(nMode:=ModeGpa.MODE_I);
	algoritms.F1_1.CanRun :=TRUE;
	F1_1_start.run ();
	Start_Prov_Pusk.reset ();
ELSIF	(Start_Prov_Pusk.answer=Answers.ANS_NO) THEN
		algoritms.F1_1.CanRun :=FALSE;
		Start_Prov_Pusk.reset ();
		reset ();
		
END_IF

IF	F1_1_start.top 	THEN
	algoritms.F1_2.CanRun :=TRUE;
	F1_2_start.run ();
END_IF
IF	F1_2_start.top AND algoritms.ppu.ppuSecond_I THEN
	algoritms.F2_R.CanRun :=TRUE;
	F2_Start.run ();
END_IF
IF	F2_start.top AND algoritms.ppu.ppuThird THEN
	algoritms.F3.CanRun :=TRUE;
	F3_Start.run ();
END_IF
IF	F3_start.top AND  algoritms.ppu.ppuForth AND NOT F4_Start.start THEN
	F4_Start_Q.ask ();
ELSE
	F4_Start_Q.reset();
END_IF
IF	F4_Start_Q.answer = Answers.ANS_YES THEN
	F4_Start_Q.reset();
	algoritms.F4.CanRun :=TRUE;
	F4_Start.run ();
	reset ();
END_IF;

METHOD PUBLIC reset
VAR_INPUT
END_VAR
SUPER^.reset();
Start_Prov_Pusk.reset ();
F4_Start_Q.reset ();
END_METHOD

END_FUNCTION_BLOCK

// K2/std12k5/Start_ALG/Start_Prov_I
{attribute 'symbol' := 'none'}
FUNCTION_BLOCK Start_Prov_I EXTENDS StepBySteapAlgoritm
VAR_INPUT
END_VAR
VAR_OUTPUT
	{attribute 'symbol' := 'read'}
	Start_Prov_Pusk:		Question(table:=ADR(ObjectTable)):=			(AnswerVariants:=(Answers.ANS_YES OR Answers.ANS_NO));
	{attribute 'symbol' := 'read'}
	F4_Start_Q:		Question(table:=ADR(ObjectTable)):=			(AnswerVariants:=Answers.ANS_YES);
END_VAR
VAR
	F1_1_start:	ph_algoritm (table:=ADR(phasesTable)):=		(phaseNumber:=0, Im:=algoritms.F1_1 , act:=PhaseAlgoritmAction.run, waitCompletion:=TRUE);
	F1_2_start:	ph_algoritm (table:=ADR(phasesTable)):=		(phaseNumber:=1, Im:=algoritms.F1_2 , act:=PhaseAlgoritmAction.run, waitCompletion:=TRUE);
	F2_Start: ph_algoritm (table:=ADR(phasesTable)):=		(phaseNumber:=2, Im:=algoritms.F2_R , act:=PhaseAlgoritmAction.run, waitCompletion:=TRUE);
	F3_Start: ph_algoritm (table:=ADR(phasesTable)):=		(phaseNumber:=3, Im:=algoritms.F3 , act:=PhaseAlgoritmAction.run, waitCompletion:=TRUE);
	F4_Start: ph_algoritm (table:=ADR(phasesTable)):=		(phaseNumber:=4, Im:=algoritms.F4 , act:=PhaseAlgoritmAction.run, waitCompletion:=TRUE);
END_VAR

SUPER^();
IF	NOT F1_1_start.start THEN
	Start_Prov_Pusk.ask ();
END_IF
IF	(Start_Prov_Pusk.answer=Answers.ANS_YES) THEN
	algManager.setMode(nMode:=ModeGpa.MODE_I);
	algoritms.F1_1.CanRun :=TRUE;
	F1_1_start.run ();
	Start_Prov_Pusk.reset ();
ELSIF	(Start_Prov_Pusk.answer=Answers.ANS_NO) THEN
		algoritms.F1_1.CanRun :=FALSE;
		Start_Prov_Pusk.reset ();
		reset ();
		
END_IF

IF	F1_1_start.top 	THEN
	algoritms.F1_2.CanRun :=TRUE;
	F1_2_start.run ();
END_IF
IF	F1_2_start.top AND algoritms.ppu.ppuSecond_I THEN
	algoritms.F2_R.CanRun :=TRUE;
	F2_Start.run ();
END_IF
IF	F2_start.top AND algoritms.ppu.ppuThird THEN
	algoritms.F3.CanRun :=TRUE;
	F3_Start.run ();
END_IF
IF	F3_start.top AND  algoritms.ppu.ppuForth AND NOT F4_Start.start THEN
	F4_Start_Q.ask ();
ELSE
	F4_Start_Q.reset();
END_IF
IF	F4_Start_Q.answer = Answers.ANS_YES THEN
	F4_Start_Q.reset();
	algoritms.F4.CanRun :=TRUE;
	F4_Start.run ();
	reset ();
END_IF;

METHOD PUBLIC reset
VAR_INPUT
END_VAR
SUPER^.reset();
Start_Prov_Pusk.reset ();
F4_Start_Q.reset ();
END_METHOD

END_FUNCTION_BLOCK

// K1/std12k5/Start_ALG/Start_Prov_k
{attribute 'symbol' := 'none'}
FUNCTION_BLOCK Start_Prov_k EXTENDS StepBySteapAlgoritm
VAR_INPUT
END_VAR
VAR_OUTPUT
	{attribute 'symbol' := 'read'}
	Start_Prov_Pusk:		Question(table:=ADR(ObjectTable)):=			(AnswerVariants:=(Answers.ANS_YES OR Answers.ANS_NO));
	{attribute 'symbol' := 'read'}
	F4_Start_Q:		Question(table:=ADR(ObjectTable)):=			(AnswerVariants:=Answers.ANS_YES);
END_VAR
VAR
	F1_1_start:	ph_algoritm (table:=ADR(phasesTable)):=		(phaseNumber:=0, Im:=algoritms.F1_1, act:=PhaseAlgoritmAction.run, waitCompletion:=TRUE);
	F1_2_start: 	ph_algoritm (table:=ADR(phasesTable)):=	(phaseNumber:=1, Im:=algoritms.F1_2, act:=PhaseAlgoritmAction.run, waitCompletion:=TRUE);
	F3_start: 	ph_algoritm (table:=ADR(phasesTable)):=		(phaseNumber:=2, Im:=algoritms.F3, act:=PhaseAlgoritmAction.run, waitCompletion:=TRUE);
	F4_Start: ph_algoritm (table:=ADR(phasesTable)):=		(phaseNumber:=4, Im:=algoritms.F4  , act:=PhaseAlgoritmAction.run, waitCompletion:=TRUE);
END_VAR

SUPER^();
IF	NOT F1_1_start.start THEN
	Start_Prov_Pusk.ask ();
END_IF
IF	(Start_Prov_Pusk.answer=Answers.ANS_YES) THEN
	algoritms.F1_1.CanRun :=TRUE;
	F1_1_start.run ();
	Start_Prov_Pusk.reset ();
	algManager.setMode(nMode:=ModeGpa.MODE_PUSKK);
ELSIF	(Start_Prov_Pusk.answer=Answers.ANS_NO) THEN
		Start_Prov_Pusk.reset ();
		algoritms.F1_1.CanRun :=FALSE;
		reset ();
END_IF
IF 	F1_1_start.top THEN
	algoritms.F1_2.CanRun :=TRUE;
	F1_2_start.run ();
END_IF
IF 	F1_2_start.top AND algoritms.ppu.ppuThird THEN
	algoritms.F3.CanRun :=TRUE;
	F3_start.run ();
END_IF
IF 	F3_start.top AND algoritms.ppu.ppuForth AND NOT F4_Start.start  THEN
	F4_Start_Q.ask ();
ELSE
	F4_Start_Q.reset ();
END_IF
IF	(F4_Start_Q.answer = Answers.ANS_YES) THEN
	F4_Start_Q.reset ();
	algoritms.F4.CanRun :=TRUE;
	F4_Start.run ();
	reset ();
END_IF;

METHOD PUBLIC reset
VAR_INPUT
END_VAR
SUPER^.reset();
Start_Prov_Pusk.reset ();
F4_Start_Q.reset ();
END_METHOD

END_FUNCTION_BLOCK

// K2/std12k5/Start_ALG/Start_Prov_k
{attribute 'symbol' := 'none'}
FUNCTION_BLOCK Start_Prov_k EXTENDS StepBySteapAlgoritm
VAR_INPUT
END_VAR
VAR_OUTPUT
	{attribute 'symbol' := 'read'}
	Start_Prov_Pusk:		Question(table:=ADR(ObjectTable)):=			(AnswerVariants:=(Answers.ANS_YES OR Answers.ANS_NO));
	{attribute 'symbol' := 'read'}
	F4_Start_Q:		Question(table:=ADR(ObjectTable)):=			(AnswerVariants:=Answers.ANS_YES);
END_VAR
VAR
	F1_1_start:	ph_algoritm (table:=ADR(phasesTable)):=		(phaseNumber:=0, Im:=algoritms.F1_1, act:=PhaseAlgoritmAction.run, waitCompletion:=TRUE);
	F1_2_start: 	ph_algoritm (table:=ADR(phasesTable)):=	(phaseNumber:=1, Im:=algoritms.F1_2, act:=PhaseAlgoritmAction.run, waitCompletion:=TRUE);
	F3_start: 	ph_algoritm (table:=ADR(phasesTable)):=		(phaseNumber:=2, Im:=algoritms.F3, act:=PhaseAlgoritmAction.run, waitCompletion:=TRUE);
	F4_Start: ph_algoritm (table:=ADR(phasesTable)):=		(phaseNumber:=4, Im:=algoritms.F4  , act:=PhaseAlgoritmAction.run, waitCompletion:=TRUE);
END_VAR

SUPER^();
IF	NOT F1_1_start.start THEN
	Start_Prov_Pusk.ask ();
END_IF
IF	(Start_Prov_Pusk.answer=Answers.ANS_YES) THEN
	algoritms.F1_1.CanRun :=TRUE;
	F1_1_start.run ();
	Start_Prov_Pusk.reset ();
	algManager.setMode(nMode:=ModeGpa.MODE_PUSKK);
ELSIF	(Start_Prov_Pusk.answer=Answers.ANS_NO) THEN
		Start_Prov_Pusk.reset ();
		algoritms.F1_1.CanRun :=FALSE;
		reset ();
END_IF
IF 	F1_1_start.top THEN
	algoritms.F1_2.CanRun :=TRUE;
	F1_2_start.run ();
END_IF
IF 	F1_2_start.top AND algoritms.ppu.ppuThird THEN
	algoritms.F3.CanRun :=TRUE;
	F3_start.run ();
END_IF
IF 	F3_start.top AND algoritms.ppu.ppuForth AND NOT F4_Start.start  THEN
	F4_Start_Q.ask ();
ELSE
	F4_Start_Q.reset ();
END_IF
IF	(F4_Start_Q.answer = Answers.ANS_YES) THEN
	F4_Start_Q.reset ();
	algoritms.F4.CanRun :=TRUE;
	F4_Start.run ();
	reset ();
END_IF;

METHOD PUBLIC reset
VAR_INPUT
END_VAR
SUPER^.reset();
Start_Prov_Pusk.reset ();
F4_Start_Q.reset ();
END_METHOD

END_FUNCTION_BLOCK

// LowLevel_Algoritms/im/Krans_Sdvig_kr4
{attribute 'symbol' := 'none'}
FUNCTION_BLOCK Krans_Sdvig_kr4 EXTENDS BaseIm
VAR_INPUT
	Krans:REFERENCE TO Kran;
	block:REFERENCE TO DiscretParametr(*(table:=ADR(objectTable))*);
	block_from_alg:REFERENCE TO DiscretParametr;
END_VAR
VAR_OUTPUT
END_VAR
VAR
	Kran_state:statusDualInput;
	Trig:R_TRIG;
END_VAR

SUPER^();
Trig (clk:=((block.Value = 1) OR (block_from_alg.Value = 1)));
IF __ISVALIDREF(Krans) THEN
	IF (krans.onStatus <> Kran_state) AND krans.sdvig AND  (block.Value = 0) AND (block_from_alg.Value = 0)	THEN
		statusSet.setBit (bitNum:=0,value:=1);
		IF	Kran_state = statusDualInput.status_on THEN
			Krans.on ();
		END_IF
		IF	Kran_state = statusDualInput.status_off THEN
			Krans.off ();
		END_IF
	ELSE 
		statusSet.setBit (bitNum:=0,value:=0);
		IF	(Trig.Q) THEN
			Kran_state:=krans.onStatus;
			krans.reset ();
		END_IF
	END_IF
	IF	(krans.onStatus = statusDualInput.status_on)  OR (krans.onStatus = statusDualInput.status_off) THEN
		Kran_state:=krans.onStatus;
	END_IF;
END_IF

END_FUNCTION_BLOCK

// K1/std12k5/Start_ALG/Start_Prov_Pms
	{attribute 'symbol' := 'none'}
FUNCTION_BLOCK Start_Prov_Pms EXTENDS StepBySteapAlgoritm
VAR_INPUT
END_VAR
VAR_OUTPUT
		{attribute 'symbol' := 'read'}
	Start_Prov_Pusk:		Question(table:=ADR(ObjectTable)):=			(AnswerVariants:=(Answers.ANS_YES OR Answers.ANS_NO));
END_VAR
VAR
	F1_start:	ph_algoritm (table:=ADR(phasesTable)):=		(phaseNumber:=0, Im:=algoritms.F1_1 , act:=PhaseAlgoritmAction.run, waitCompletion:=TRUE);
	P_ms_start: ph_algoritm (table:=ADR(phasesTable)):=		(phaseNumber:=1, Im:=algoritms.Pms , act:=PhaseAlgoritmAction.run, waitCompletion:=TRUE);
END_VAR

SUPER^();
IF	NOT F1_start.start THEN
	Start_Prov_Pusk.ask ();
END_IF
IF	(Start_Prov_Pusk.answer=Answers.ANS_YES) THEN
	algManager.setMode(nMode:=ModeGpa.MODE_PROVPMS);
	algoritms.F1_1.CanRun :=TRUE;
	F1_start.run ();
	Start_Prov_Pusk.reset ();
ELSIF	(Start_Prov_Pusk.answer=Answers.ANS_NO) THEN
		algoritms.F1_1.CanRun :=FALSE;
		Start_Prov_Pusk.reset ();
		reset ();
END_IF
IF 	F1_start.top THEN
	algoritms.Pms.CanRun:=TRUE;
	P_ms_start.run ();
	reset ();
END_IF

METHOD PUBLIC reset
VAR_INPUT
END_VAR
SUPER^.reset();
Start_Prov_Pusk.reset ();
END_METHOD

END_FUNCTION_BLOCK

// K2/std12k5/Start_ALG/Start_Prov_Pms
	{attribute 'symbol' := 'none'}
FUNCTION_BLOCK Start_Prov_Pms EXTENDS StepBySteapAlgoritm
VAR_INPUT
END_VAR
VAR_OUTPUT
		{attribute 'symbol' := 'read'}
	Start_Prov_Pusk:		Question(table:=ADR(ObjectTable)):=			(AnswerVariants:=(Answers.ANS_YES OR Answers.ANS_NO));
END_VAR
VAR
	F1_start:	ph_algoritm (table:=ADR(phasesTable)):=		(phaseNumber:=0, Im:=algoritms.F1_1 , act:=PhaseAlgoritmAction.run, waitCompletion:=TRUE);
	P_ms_start: ph_algoritm (table:=ADR(phasesTable)):=		(phaseNumber:=1, Im:=algoritms.Pms , act:=PhaseAlgoritmAction.run, waitCompletion:=TRUE);
END_VAR

SUPER^();
IF	NOT F1_start.start THEN
	Start_Prov_Pusk.ask ();
END_IF
IF	(Start_Prov_Pusk.answer=Answers.ANS_YES) THEN
	algManager.setMode(nMode:=ModeGpa.MODE_PROVPMS);
	algoritms.F1_1.CanRun :=TRUE;
	F1_start.run ();
	Start_Prov_Pusk.reset ();
ELSIF	(Start_Prov_Pusk.answer=Answers.ANS_NO) THEN
		algoritms.F1_1.CanRun :=FALSE;
		Start_Prov_Pusk.reset ();
		reset ();
END_IF
IF 	F1_start.top THEN
	algoritms.Pms.CanRun:=TRUE;
	P_ms_start.run ();
	reset ();
END_IF

METHOD PUBLIC reset
VAR_INPUT
END_VAR
SUPER^.reset();
Start_Prov_Pusk.reset ();
END_METHOD

END_FUNCTION_BLOCK

// K1/std12k5/Start_ALG/Start_Prov_V
{attribute 'symbol' := 'none'}
FUNCTION_BLOCK Start_Prov_V EXTENDS StepBySteapAlgoritm
VAR_INPUT
END_VAR
VAR_OUTPUT
	{attribute 'symbol' := 'read'}
	Start_Prov_Pusk:		Question(table:=ADR(ObjectTable)):=			(AnswerVariants:=(Answers.ANS_YES OR Answers.ANS_NO));
	{attribute 'symbol' := 'read'}
	Ypr_MV:		Question(table:=ADR(ObjectTable)):=			(AnswerVariants:=Answers.ANS_YES);
END_VAR
VAR
	F1_start:	ph_algoritm (table:=ADR(phasesTable)):=		(phaseNumber:=0, Im:=algoritms.F1_1, act:=PhaseAlgoritmAction.run, waitCompletion:=TRUE);
	F2ch_start: 	ph_algoritm (table:=ADR(phasesTable)):=		(phaseNumber:=1, Im:=algoritms.F2_Ch, act:=PhaseAlgoritmAction.run, waitCompletion:=TRUE);
	F2r_start: 	ph_algoritm (table:=ADR(phasesTable)):=		(phaseNumber:=2, Im:=algoritms.F2_R, act:=PhaseAlgoritmAction.run, waitCompletion:=TRUE);
	Prov_MV:	CustomPhase (table:=ADR(phasesTable)):=			(phaseNumber:=3);
END_VAR

SUPER^();
IF	NOT F1_start.start THEN
	Start_Prov_Pusk.ask ();
END_IF

IF	(Start_Prov_Pusk.answer=Answers.ANS_YES) THEN
	algoritms.F1_1.CanRun :=TRUE;
	F1_start.run ();
	Start_Prov_Pusk.reset ();
	IF 	algoritms.ppu.ppuFirst_for_V_Ch THEN
		algManager.setMode(nMode:=ModeGpa.MODE_PUSKV_Ch);
	END_IF
	IF 	algoritms.ppu.ppuFirst_for_V_r  THEN
		algManager.setMode(nMode:=ModeGpa.MODE_PUSKV_r);
	END_IF;
ELSIF	(Start_Prov_Pusk.answer=Answers.ANS_NO) THEN
		algoritms.F1_1.CanRun :=FALSE;
		Start_Prov_Pusk.reset ();
		reset ();
END_IF
IF 	F1_start.top AND algoritms.ppu.ppuSecond_V_Pusk_Ch AND NOT (F2ch_start.start) AND (algmanager.mode = modegpa.MODE_PUSKV_Ch) THEN
	algoritms.F2_Ch.CanRun:=TRUE;
	F2ch_start.run ();
END_IF
IF 	F1_start.top AND algoritms.ppu.ppuSecond_V_Pusk_R AND NOT (F2r_start.start ) AND (algmanager.mode = modegpa.MODE_PUSKV_R) THEN
	algoritms.F2_R.CanRun:=TRUE;
	F2r_start.run ();
END_IF
IF	(F2ch_start.top OR F2r_start.top) AND NOT Prov_MV.top THEN
	Ypr_MV.ask ();
	Prov_MV.top:=TRUE;
END_IF
IF	(Ypr_MV.answer=Answers.ANS_YES) THEN
	Ypr_MV.reset ();
	im.mv.EnableOpcControl();
	end ();
END_IF

METHOD PUBLIC reset
VAR_INPUT
END_VAR
SUPER^.reset();
Start_Prov_Pusk.reset ();
Ypr_MV.reset();
im.mv.DisableOpcControl	();
END_METHOD

END_FUNCTION_BLOCK

// K2/std12k5/Start_ALG/Start_Prov_V
{attribute 'symbol' := 'none'}
FUNCTION_BLOCK Start_Prov_V EXTENDS StepBySteapAlgoritm
VAR_INPUT
END_VAR
VAR_OUTPUT
	{attribute 'symbol' := 'read'}
	Start_Prov_Pusk:		Question(table:=ADR(ObjectTable)):=			(AnswerVariants:=(Answers.ANS_YES OR Answers.ANS_NO));
	{attribute 'symbol' := 'read'}
	Ypr_MV:		Question(table:=ADR(ObjectTable)):=			(AnswerVariants:=Answers.ANS_YES);
END_VAR
VAR
	F1_start:	ph_algoritm (table:=ADR(phasesTable)):=		(phaseNumber:=0, Im:=algoritms.F1_1, act:=PhaseAlgoritmAction.run, waitCompletion:=TRUE);
	F2ch_start: 	ph_algoritm (table:=ADR(phasesTable)):=		(phaseNumber:=1, Im:=algoritms.F2_Ch, act:=PhaseAlgoritmAction.run, waitCompletion:=TRUE);
	F2r_start: 	ph_algoritm (table:=ADR(phasesTable)):=		(phaseNumber:=2, Im:=algoritms.F2_R, act:=PhaseAlgoritmAction.run, waitCompletion:=TRUE);
	Prov_MV:	CustomPhase (table:=ADR(phasesTable)):=			(phaseNumber:=3);
END_VAR

SUPER^();
IF	NOT F1_start.start THEN
	Start_Prov_Pusk.ask ();
END_IF

IF	(Start_Prov_Pusk.answer=Answers.ANS_YES) THEN
	algoritms.F1_1.CanRun :=TRUE;
	F1_start.run ();
	Start_Prov_Pusk.reset ();
	IF 	algoritms.ppu.ppuFirst_for_V_Ch THEN
		algManager.setMode(nMode:=ModeGpa.MODE_PUSKV_Ch);
	END_IF
	IF 	algoritms.ppu.ppuFirst_for_V_r  THEN
		algManager.setMode(nMode:=ModeGpa.MODE_PUSKV_r);
	END_IF;
ELSIF	(Start_Prov_Pusk.answer=Answers.ANS_NO) THEN
		algoritms.F1_1.CanRun :=FALSE;
		Start_Prov_Pusk.reset ();
		reset ();
END_IF
IF 	F1_start.top AND algoritms.ppu.ppuSecond_V_Pusk_Ch AND NOT (F2ch_start.start) AND (algmanager.mode = modegpa.MODE_PUSKV_Ch) THEN
	algoritms.F2_Ch.CanRun:=TRUE;
	F2ch_start.run ();
END_IF
IF 	F1_start.top AND algoritms.ppu.ppuSecond_V_Pusk_R AND NOT (F2r_start.start ) AND (algmanager.mode = modegpa.MODE_PUSKV_R) THEN
	algoritms.F2_R.CanRun:=TRUE;
	F2r_start.run ();
END_IF
IF	(F2ch_start.top OR F2r_start.top) AND NOT Prov_MV.top THEN
	Ypr_MV.ask ();
	Prov_MV.top:=TRUE;
END_IF
IF	(Ypr_MV.answer=Answers.ANS_YES) THEN
	Ypr_MV.reset ();
	im.mv.EnableOpcControl();
	end ();
END_IF

METHOD PUBLIC reset
VAR_INPUT
END_VAR
SUPER^.reset();
Start_Prov_Pusk.reset ();
Ypr_MV.reset();
im.mv.DisableOpcControl	();
END_METHOD

END_FUNCTION_BLOCK

// K1/std12k5/Start_ALG/Start_Pusk_AP
{attribute 'symbol' := 'none'}
FUNCTION_BLOCK Start_Pusk_AP EXTENDS StepBySteapAlgoritm
VAR_INPUT
END_VAR
VAR_OUTPUT
	{attribute 'symbol' := 'read'}
	Start_Prov_Pusk:		Question(table:=ADR(ObjectTable)):=			(AnswerVariants:=(Answers.ANS_YES OR Answers.ANS_NO));
END_VAR
VAR
	F1_1_start:	ph_algoritm (table:=ADR(phasesTable)):=		(phaseNumber:=0, Im:=algoritms.F1_1 , act:=PhaseAlgoritmAction.run, waitCompletion:=TRUE);
	F2ch_start:	ph_algoritm (table:=ADR(phasesTable)):=		(phaseNumber:=1, Im:=algoritms.F2_Ch	 , act:=PhaseAlgoritmAction.run, waitCompletion:=TRUE);
	F2r_Start: ph_algoritm (table:=ADR(phasesTable)):=		(phaseNumber:=2, Im:=algoritms.F2_r , act:=PhaseAlgoritmAction.run, waitCompletion:=TRUE);
	F3_Start: ph_algoritm (table:=ADR(phasesTable)):=		(phaseNumber:=3, Im:=algoritms.F3 , act:=PhaseAlgoritmAction.run, waitCompletion:=TRUE);
	F4_Start: ph_algoritm (table:=ADR(phasesTable)):=		(phaseNumber:=4, Im:=algoritms.F4 , act:=PhaseAlgoritmAction.run, waitCompletion:=TRUE);
END_VAR

SUPER^();
IF	NOT F1_1_start.start THEN
	Start_Prov_Pusk.ask ();
END_IF
IF	(Start_Prov_Pusk.answer=Answers.ANS_YES) THEN
	IF 	algoritms.ppu.ppuFirst_for_Pusk_Ch THEN
		algManager.setMode(nMode:=ModeGpa.MODE_PUSKAP_Ch);
	END_IF
	IF 	algoritms.ppu.ppuFirst_for_Pusk_r THEN
		algManager.setMode(nMode:=ModeGpa.MODE_PUSKAP_r);
	END_IF
	algoritms.F1_1.CanRun :=TRUE;
	F1_1_start.run ();
	Start_Prov_Pusk.reset ();
ELSIF	(Start_Prov_Pusk.answer=Answers.ANS_NO) THEN
		algoritms.F1_1.CanRun :=FALSE;
		Start_Prov_Pusk.reset ();
		reset ();
END_IF


IF	F1_1_start.top AND algoritms.ppu.ppuSecond_V_Pusk_Ch AND (NOT (F2ch_start.start)) AND (algmanager.mode = modegpa.MODE_PUSKAP_Ch) THEN
	algoritms.F2_Ch.CanRun:=TRUE;
	F2ch_start.run ();
END_IF
IF	F1_1_start.top AND algoritms.ppu.ppuSecond_V_Pusk_R AND (NOT ( F2r_Start.start)) AND (algmanager.mode = modegpa.MODE_PUSKAP_R) THEN
	algoritms.F2_R.CanRun:=TRUE;
	F2r_start.run ();
END_IF
IF	(F2ch_start.top OR F2r_start.top) AND algoritms.ppu.ppuThird THEN
	algoritms.F3.CanRun:=TRUE;
	F3_Start.run ();
END_IF
IF	F3_start.top AND  algoritms.ppu.ppuForth THEN
	algoritms.F4.CanRun:=TRUE;
	F4_Start.run ();
	reset ();
END_IF

METHOD PUBLIC reset
VAR_INPUT
END_VAR
SUPER^.reset();
Start_Prov_Pusk.reset ();
END_METHOD

END_FUNCTION_BLOCK

// K2/std12k5/Start_ALG/Start_Pusk_AP
{attribute 'symbol' := 'none'}
FUNCTION_BLOCK Start_Pusk_AP EXTENDS StepBySteapAlgoritm
VAR_INPUT
END_VAR
VAR_OUTPUT
	{attribute 'symbol' := 'read'}
	Start_Prov_Pusk:		Question(table:=ADR(ObjectTable)):=			(AnswerVariants:=(Answers.ANS_YES OR Answers.ANS_NO));
END_VAR
VAR
	F1_1_start:	ph_algoritm (table:=ADR(phasesTable)):=		(phaseNumber:=0, Im:=algoritms.F1_1 , act:=PhaseAlgoritmAction.run, waitCompletion:=TRUE);
	F2ch_start:	ph_algoritm (table:=ADR(phasesTable)):=		(phaseNumber:=1, Im:=algoritms.F2_Ch	 , act:=PhaseAlgoritmAction.run, waitCompletion:=TRUE);
	F2r_Start: ph_algoritm (table:=ADR(phasesTable)):=		(phaseNumber:=2, Im:=algoritms.F2_r , act:=PhaseAlgoritmAction.run, waitCompletion:=TRUE);
	F3_Start: ph_algoritm (table:=ADR(phasesTable)):=		(phaseNumber:=3, Im:=algoritms.F3 , act:=PhaseAlgoritmAction.run, waitCompletion:=TRUE);
	F4_Start: ph_algoritm (table:=ADR(phasesTable)):=		(phaseNumber:=4, Im:=algoritms.F4 , act:=PhaseAlgoritmAction.run, waitCompletion:=TRUE);
END_VAR

SUPER^();
IF	NOT F1_1_start.start THEN
	Start_Prov_Pusk.ask ();
END_IF
IF	(Start_Prov_Pusk.answer=Answers.ANS_YES) THEN
	IF 	algoritms.ppu.ppuFirst_for_Pusk_Ch THEN
		algManager.setMode(nMode:=ModeGpa.MODE_PUSKAP_Ch);
	END_IF
	IF 	algoritms.ppu.ppuFirst_for_Pusk_r THEN
		algManager.setMode(nMode:=ModeGpa.MODE_PUSKAP_r);
	END_IF
	algoritms.F1_1.CanRun :=TRUE;
	F1_1_start.run ();
	Start_Prov_Pusk.reset ();
ELSIF	(Start_Prov_Pusk.answer=Answers.ANS_NO) THEN
		algoritms.F1_1.CanRun :=FALSE;
		Start_Prov_Pusk.reset ();
		reset ();
END_IF


IF	F1_1_start.top AND algoritms.ppu.ppuSecond_V_Pusk_Ch AND (NOT (F2ch_start.start)) AND (algmanager.mode = modegpa.MODE_PUSKAP_Ch) THEN
	algoritms.F2_Ch.CanRun:=TRUE;
	F2ch_start.run ();
END_IF
IF	F1_1_start.top AND algoritms.ppu.ppuSecond_V_Pusk_R AND (NOT ( F2r_Start.start)) AND (algmanager.mode = modegpa.MODE_PUSKAP_R) THEN
	algoritms.F2_R.CanRun:=TRUE;
	F2r_start.run ();
END_IF
IF	(F2ch_start.top OR F2r_start.top) AND algoritms.ppu.ppuThird THEN
	algoritms.F3.CanRun:=TRUE;
	F3_Start.run ();
END_IF
IF	F3_start.top AND  algoritms.ppu.ppuForth THEN
	algoritms.F4.CanRun:=TRUE;
	F4_Start.run ();
	reset ();
END_IF

METHOD PUBLIC reset
VAR_INPUT
END_VAR
SUPER^.reset();
Start_Prov_Pusk.reset ();
END_METHOD

END_FUNCTION_BLOCK

// K1/std12k5/Start_ALG/Start_Pusk_PP
{attribute 'symbol' := 'none'}
FUNCTION_BLOCK Start_Pusk_PP EXTENDS StepBySteapAlgoritm
VAR_INPUT
END_VAR
	
VAR_OUTPUT
	{attribute 'symbol' := 'read'}
	Start_Prov_Pusk:		Question(table:=ADR(ObjectTable)):=			(AnswerVariants:=(Answers.ANS_YES OR Answers.ANS_NO));
	{attribute 'symbol' := 'read'}
	F2_Ask:		Question(table:=ADR(ObjectTable)):=			(AnswerVariants:=Answers.ANS_YES);
	{attribute 'symbol' := 'read'}
	F3_Ask:		Question(table:=ADR(ObjectTable)):=			(AnswerVariants:=Answers.ANS_YES);
	{attribute 'symbol' := 'read'}
	F4_Ask:		Question(table:=ADR(ObjectTable)):=			(AnswerVariants:=Answers.ANS_YES);
END_VAR
VAR
	F1_1_start:	ph_algoritm (table:=ADR(phasesTable)):=		(phaseNumber:=0, Im:=algoritms.F1_1 , act:=PhaseAlgoritmAction.run, waitCompletion:=TRUE);
	F2ch_start:	ph_algoritm (table:=ADR(phasesTable)):=		(phaseNumber:=1, Im:=algoritms.F2_Ch , act:=PhaseAlgoritmAction.run, waitCompletion:=TRUE);
	F2r_Start: ph_algoritm (table:=ADR(phasesTable)):=		(phaseNumber:=2, Im:=algoritms.F2_R , act:=PhaseAlgoritmAction.run, waitCompletion:=TRUE);
	F3_Start: ph_algoritm (table:=ADR(phasesTable)):=		(phaseNumber:=3, Im:=algoritms.F3 , act:=PhaseAlgoritmAction.run, waitCompletion:=TRUE);
	F4_Start: ph_algoritm (table:=ADR(phasesTable)):=		(phaseNumber:=4, Im:=algoritms.F4 , act:=PhaseAlgoritmAction.run, waitCompletion:=TRUE);
END_VAR

SUPER^();

IF	NOT F1_1_start.start THEN
	Start_Prov_Pusk.ask ();
END_IF

IF	(Start_Prov_Pusk.answer=Answers.ANS_YES) THEN
	algoritms.F1_1.CanRun :=TRUE;
	IF 	algoritms.ppu.ppuFirst_for_Pusk_Ch THEN
		algManager.setMode(nMode:=ModeGpa.MODE_PUSKPP_Ch);
	END_IF
	IF 	algoritms.ppu.ppuFirst_for_Pusk_r THEN
		algManager.setMode(nMode:=ModeGpa.MODE_PUSKPP_r);
	END_IF
	F1_1_start.run ();
	Start_Prov_Pusk.reset ();
ELSIF	(Start_Prov_Pusk.answer=Answers.ANS_NO) THEN
		algoritms.F1_1.CanRun :=FALSE;
		Start_Prov_Pusk.reset ();
		reset ();
END_IF
///////////////////////////////////////////////////
IF	F1_1_start.top AND ((algoritms.ppu.ppuSecond_V_Pusk_Ch AND (algmanager.mode = modegpa.MODE_PUSKPP_Ch) AND NOT (F2ch_start.start)) OR 
	(algoritms.ppu.ppuSecond_V_Pusk_r AND (algmanager.mode = modegpa.MODE_PUSKPP_r)	AND NOT (F2r_start.start))) THEN
	F2_Ask.ask ();
ELSE
	F2_Ask.reset ();
END_IF
///////////////////////////////////////////////////
IF	(F2_Ask.answer=Answers.ANS_YES) THEN
	F2_Ask.reset ();
	IF	(algmanager.mode = modegpa.MODE_PUSKPP_Ch) AND (algoritms.ppu.ppuSecond_V_Pusk_Ch) THEN
		algoritms.F2_Ch.canrun:=TRUE;
		F2ch_start.run ();
	END_IF;
	IF	(algmanager.mode = modegpa.MODE_PUSKPP_r) AND algoritms.ppu.ppuSecond_V_Pusk_r THEN
		algoritms.F2_r.canrun:=TRUE;
		F2r_start.run ();
	END_IF;
	
END_IF
///////////////////////////////////////////////////
IF	(F2ch_start.top OR F2r_start.top) AND algoritms.ppu.ppuThird AND NOT F3_Start.start THEN
	F3_Ask.ask ();
ELSE
	F3_Ask.reset ();
END_IF
///////////////////////////////////////////////////
IF	(F3_Ask.answer=Answers.ANS_YES) AND algoritms.ppu.ppuThird THEN
	algoritms.F3.CanRun:=TRUE;
	F3_Ask.reset ();
	F3_Start.run ();
END_IF
///////////////////////////////////////////////////
IF	F3_Start.top AND algoritms.ppu.ppuForth AND NOT F4_Start.start THEN
	F4_Ask.ask ();
ELSE
	F4_Ask.reset ();
END_IF
///////////////////////////////////////////////////
IF	(F4_Ask.answer=Answers.ANS_YES) AND algoritms.ppu.ppuForth THEN
	F4_Ask.reset ();
	algoritms.F4.CanRun:=TRUE;
	F4_Start.run ();
	reset ();
END_IF

METHOD PUBLIC reset
VAR_INPUT
END_VAR
SUPER^.reset();
Start_Prov_Pusk.reset ();
F2_Ask.reset ();
F3_Ask.reset ();
F4_Ask.reset ();
END_METHOD

END_FUNCTION_BLOCK

// K2/std12k5/Start_ALG/Start_Pusk_PP
{attribute 'symbol' := 'none'}
FUNCTION_BLOCK Start_Pusk_PP EXTENDS StepBySteapAlgoritm
VAR_INPUT
END_VAR
	
VAR_OUTPUT
	{attribute 'symbol' := 'read'}
	Start_Prov_Pusk:		Question(table:=ADR(ObjectTable)):=			(AnswerVariants:=(Answers.ANS_YES OR Answers.ANS_NO));
	{attribute 'symbol' := 'read'}
	F2_Ask:		Question(table:=ADR(ObjectTable)):=			(AnswerVariants:=Answers.ANS_YES);
	{attribute 'symbol' := 'read'}
	F3_Ask:		Question(table:=ADR(ObjectTable)):=			(AnswerVariants:=Answers.ANS_YES);
	{attribute 'symbol' := 'read'}
	F4_Ask:		Question(table:=ADR(ObjectTable)):=			(AnswerVariants:=Answers.ANS_YES);
END_VAR
VAR
	F1_1_start:	ph_algoritm (table:=ADR(phasesTable)):=		(phaseNumber:=0, Im:=algoritms.F1_1 , act:=PhaseAlgoritmAction.run, waitCompletion:=TRUE);
	F2ch_start:	ph_algoritm (table:=ADR(phasesTable)):=		(phaseNumber:=1, Im:=algoritms.F2_Ch , act:=PhaseAlgoritmAction.run, waitCompletion:=TRUE);
	F2r_Start: ph_algoritm (table:=ADR(phasesTable)):=		(phaseNumber:=2, Im:=algoritms.F2_R , act:=PhaseAlgoritmAction.run, waitCompletion:=TRUE);
	F3_Start: ph_algoritm (table:=ADR(phasesTable)):=		(phaseNumber:=3, Im:=algoritms.F3 , act:=PhaseAlgoritmAction.run, waitCompletion:=TRUE);
	F4_Start: ph_algoritm (table:=ADR(phasesTable)):=		(phaseNumber:=4, Im:=algoritms.F4 , act:=PhaseAlgoritmAction.run, waitCompletion:=TRUE);
END_VAR

SUPER^();

IF	NOT F1_1_start.start THEN
	Start_Prov_Pusk.ask ();
END_IF

IF	(Start_Prov_Pusk.answer=Answers.ANS_YES) THEN
	algoritms.F1_1.CanRun :=TRUE;
	IF 	algoritms.ppu.ppuFirst_for_Pusk_Ch THEN
		algManager.setMode(nMode:=ModeGpa.MODE_PUSKPP_Ch);
	END_IF
	IF 	algoritms.ppu.ppuFirst_for_Pusk_r THEN
		algManager.setMode(nMode:=ModeGpa.MODE_PUSKPP_r);
	END_IF
	F1_1_start.run ();
	Start_Prov_Pusk.reset ();
ELSIF	(Start_Prov_Pusk.answer=Answers.ANS_NO) THEN
		algoritms.F1_1.CanRun :=FALSE;
		Start_Prov_Pusk.reset ();
		reset ();
END_IF
///////////////////////////////////////////////////
IF	F1_1_start.top AND ((algoritms.ppu.ppuSecond_V_Pusk_Ch AND (algmanager.mode = modegpa.MODE_PUSKPP_Ch) AND NOT (F2ch_start.start)) OR 
	(algoritms.ppu.ppuSecond_V_Pusk_r AND (algmanager.mode = modegpa.MODE_PUSKPP_r)	AND NOT (F2r_start.start))) THEN
	F2_Ask.ask ();
ELSE
	F2_Ask.reset ();
END_IF
///////////////////////////////////////////////////
IF	(F2_Ask.answer=Answers.ANS_YES) THEN
	F2_Ask.reset ();
	IF	(algmanager.mode = modegpa.MODE_PUSKPP_Ch) AND (algoritms.ppu.ppuSecond_V_Pusk_Ch) THEN
		algoritms.F2_Ch.canrun:=TRUE;
		F2ch_start.run ();
	END_IF;
	IF	(algmanager.mode = modegpa.MODE_PUSKPP_r) AND algoritms.ppu.ppuSecond_V_Pusk_r THEN
		algoritms.F2_r.canrun:=TRUE;
		F2r_start.run ();
	END_IF;
	
END_IF
///////////////////////////////////////////////////
IF	(F2ch_start.top OR F2r_start.top) AND algoritms.ppu.ppuThird AND NOT F3_Start.start THEN
	F3_Ask.ask ();
ELSE
	F3_Ask.reset ();
END_IF
///////////////////////////////////////////////////
IF	(F3_Ask.answer=Answers.ANS_YES) AND algoritms.ppu.ppuThird THEN
	algoritms.F3.CanRun:=TRUE;
	F3_Ask.reset ();
	F3_Start.run ();
END_IF
///////////////////////////////////////////////////
IF	F3_Start.top AND algoritms.ppu.ppuForth AND NOT F4_Start.start THEN
	F4_Ask.ask ();
ELSE
	F4_Ask.reset ();
END_IF
///////////////////////////////////////////////////
IF	(F4_Ask.answer=Answers.ANS_YES) AND algoritms.ppu.ppuForth THEN
	F4_Ask.reset ();
	algoritms.F4.CanRun:=TRUE;
	F4_Start.run ();
	reset ();
END_IF

METHOD PUBLIC reset
VAR_INPUT
END_VAR
SUPER^.reset();
Start_Prov_Pusk.reset ();
F2_Ask.reset ();
F3_Ask.reset ();
F4_Ask.reset ();
END_METHOD

END_FUNCTION_BLOCK

// K1/std12k5/Start_ALG/Start_Test_IM
{attribute 'symbol' := 'none'}
FUNCTION_BLOCK Start_Test_IM EXTENDS StepBySteapAlgoritm
VAR_INPUT
END_VAR
	
VAR_OUTPUT
	{attribute 'symbol' := 'read'}
	Start_Prov_Pusk:		Question(table:=ADR(ObjectTable)):=			(AnswerVariants:=(Answers.ANS_YES OR Answers.ANS_NO));
END_VAR
VAR
	Alg_Start_reset:	ph_algoritm (table:=ADR(phasesTable)):=		(phaseNumber:=0, Im:=algoritms.Test_IM, act:=PhaseAlgoritmAction.run, waitCompletion:=FALSE);
END_VAR

SUPER^();
IF	NOT Alg_Start_reset.start THEN
	Start_Prov_Pusk.ask ();
END_IF
IF	(Start_Prov_Pusk.answer=Answers.ANS_YES) THEN
	algoritms.Test_IM.CanRun:=TRUE;
	Alg_Start_reset.run ();
	Start_Prov_Pusk.reset ();
	reset ();
ELSIF	(Start_Prov_Pusk.answer=Answers.ANS_NO) THEN
		algoritms.Test_IM.CanRun:=FALSE;
		Start_Prov_Pusk.reset ();
		reset ();
		
END_IF

METHOD PUBLIC reset
VAR_INPUT
END_VAR
SUPER^.reset();
Start_Prov_Pusk.reset ();
END_METHOD

END_FUNCTION_BLOCK

// K2/std12k5/Start_ALG/Start_Test_IM
{attribute 'symbol' := 'none'}
FUNCTION_BLOCK Start_Test_IM EXTENDS StepBySteapAlgoritm
VAR_INPUT
END_VAR
	
VAR_OUTPUT
	{attribute 'symbol' := 'read'}
	Start_Prov_Pusk:		Question(table:=ADR(ObjectTable)):=			(AnswerVariants:=(Answers.ANS_YES OR Answers.ANS_NO));
END_VAR
VAR
	Alg_Start_reset:	ph_algoritm (table:=ADR(phasesTable)):=		(phaseNumber:=0, Im:=algoritms.Test_IM, act:=PhaseAlgoritmAction.run, waitCompletion:=FALSE);
END_VAR

SUPER^();
IF	NOT Alg_Start_reset.start THEN
	Start_Prov_Pusk.ask ();
END_IF
IF	(Start_Prov_Pusk.answer=Answers.ANS_YES) THEN
	algoritms.Test_IM.CanRun:=TRUE;
	Alg_Start_reset.run ();
	Start_Prov_Pusk.reset ();
	reset ();
ELSIF	(Start_Prov_Pusk.answer=Answers.ANS_NO) THEN
		algoritms.Test_IM.CanRun:=FALSE;
		Start_Prov_Pusk.reset ();
		reset ();
		
END_IF

METHOD PUBLIC reset
VAR_INPUT
END_VAR
SUPER^.reset();
Start_Prov_Pusk.reset ();
END_METHOD

END_FUNCTION_BLOCK

// K1/std12k5/TestIm/BlockOpcControl
FUNCTION BlockOpcControl : bool
VAR_INPUT
	block:BOOL;
END_VAR
VAR
	
END_VAR

BlockIm(im:=im.kran6,block:=block);
BlockIm(im:=im.pns,block:=block);

BlockIm(im:=im.CMN,block:=block);
BlockIm(im:=im.TEN_Kollectira,block:=block);

BlockIm(im:=im.v1_Avom,block:=block);
BlockIm(im:=im.v2_Avom,block:=block);
BlockIm(im:=im.v3_Avom,block:=block);
BlockIm(im:=im.v4_Avom,block:=block);
BlockIm(im:=im.KaloriferAVOM,block:=block);

END_FUNCTION

// K2/std12k5/TestIm/BlockOpcControl
FUNCTION BlockOpcControl : BOOL
VAR_INPUT
	block:BOOL;
END_VAR
VAR
	
END_VAR

BlockIm(im:=im.kran6,block:=block);
BlockIm(im:=im.pns,block:=block);

BlockIm(im:=im.CMN,block:=block);
BlockIm(im:=im.TEN_Kollectira,block:=block);

BlockIm(im:=im.v1_Avom,block:=block);
BlockIm(im:=im.v2_Avom,block:=block);
BlockIm(im:=im.v3_Avom,block:=block);
BlockIm(im:=im.v4_Avom,block:=block);
BlockIm(im:=im.KaloriferAVOM,block:=block);

END_FUNCTION

// K1/std12k5/TestIm/TestImAlg
	{attribute 'symbol' := 'none'}
FUNCTION_BLOCK TestImAlg EXTENDS BaseAlgoritm
VAR_INPUT
END_VAR
VAR_OUTPUT
END_VAR
VAR
END_VAR

SUPER^();
BlockIm(im:=im.TEN_MB,block:=((BlockOpcControl(block:=FALSE)) OR (im.CMN.onStatus = statusDualInput.STATUS_ERROR) OR (im.CMN.onStatus = statusDualInput.STATUS_NOTDEFINED) OR 
(im.CMN.onStatus = statusDualInput.STATUS_OFF) OR (im.CMN.onStatus = statusDualInput.STATUS_TRANSITIONAL) ));
IF	(im.CMN.onStatus = statusDualInput.STATUS_OFF) AND (im.TEN_MB.onStatus = statusDualInput.STATUS_on) THEN
	im.TEN_MB.off();
END_IF
BlockIm(im:=im.nu.nu1,block:=((BlockOpcControl(block:=FALSE)) OR (im.PNS.onStatus = statusDualInput.STATUS_ERROR) OR (im.pns.onStatus = statusDualInput.STATUS_NOTDEFINED) OR 
(im.pns.onStatus = statusDualInput.STATUS_OFF) OR (im.pns.onStatus = statusDualInput.STATUS_TRANSITIONAL) ));
BlockIm(im:=im.nu.nu2,block:=((BlockOpcControl(block:=FALSE)) OR (im.PNS.onStatus = statusDualInput.STATUS_ERROR) OR (im.pns.onStatus = statusDualInput.STATUS_NOTDEFINED) OR 
(im.pns.onStatus = statusDualInput.STATUS_OFF) OR (im.pns.onStatus = statusDualInput.STATUS_TRANSITIONAL) ));
IF	(im.pns.onStatus = statusDualInput.STATUS_OFF) AND ((im.nu.nu1.onStatus = statusDualInput.STATUS_on) OR (im.nu.nu2.onStatus = statusDualInput.STATUS_on)) THEN
	im.nu.off();
END_IF

METHOD PUBLIC reset
VAR_INPUT
END_VAR
SUPER^.reset();
BlockOpcControl(block:=TRUE);
IF	(algmanager.mode <> modegpa.MODE_AO) AND (algmanager.mode <> modegpa.MODE_NO) AND (algmanager.mode <> modegpa.MODE_EO) THEN
	algManager.setMode(nMode:=ModeGpa.MODE_STOP);
END_IF
im.PNS.DisableOpcControl();
im.nu.nu1.DisableOpcControl();
im.nu.nu2.DisableOpcControl();
im.CMN.DisableOpcControl();
im.TEN_MB.DisableOpcControl();
IF	im.PNS.onStatus = statusDualInput.STATUS_ON THEN
	im.PNS.off();
END_IF
IF	im.nu.nu1.onStatus = statusDualInput.STATUS_ON THEN
	im.nu.nu1.off();
END_IF
IF	im.nu.nu2.onStatus = statusDualInput.STATUS_ON THEN
	im.nu.nu2.off();
END_IF
IF	im.cmn.onStatus = statusDualInput.STATUS_ON THEN
	im.cmn.off();
END_IF
IF	im.TEN_MB.onStatus = statusDualInput.STATUS_ON THEN
	im.TEN_MB.off();
END_IF
END_METHOD

METHOD PUBLIC run
VAR_INPUT
END_VAR
SUPER^.run();
BlockOpcControl(block:=FALSE);
algManager.setMode(nMode:=ModeGpa.MODE_TESTIM);

im.mv.DisableOpcControl ();
im.kran1.DisableOpcControl ();
im.kran2.DisableOpcControl ();
im.kran3.DisableOpcControl ();
im.kran3b.DisableOpcControl ();
im.kran4.DisableOpcControl ();
im.kran5.DisableOpcControl ();
END_METHOD

